C05467=1069.502,171.520,421.573,173.265,27.850,155.032
C05468=1069.508,171.769,421.550,173.266,27.852,155.033
C05469=1069.513,172.019,421.528,173.269,27.855,155.033
C05470=1069.519,172.267,421.505,173.270,27.858,155.034
C05471=1069.525,172.515,421.483,173.273,27.861,155.034
C05472=1069.530,172.765,421.461,173.274,27.864,155.034
C05473=1069.536,173.014,421.438,173.277,27.867,155.035
C05474=1069.542,173.263,421.416,173.278,27.870,155.035
C05475=1069.548,173.512,421.393,173.280,27.872,155.036
C05476=1069.553,173.760,421.370,173.282,27.875,155.036
C05477=1069.558,174.010,421.348,173.284,27.878,155.036
C05478=1069.565,174.258,421.326,173.286,27.881,155.037
C05479=1069.570,174.508,421.304,173.288,27.884,155.037
C05480=1069.576,174.790,421.278,173.290,27.887,155.037
C05481=1069.583,175.072,421.253,173.293,27.890,155.038
C05482=1069.590,175.355,421.226,173.295,27.893,155.038
C05483=1069.597,175.637,421.201,173.297,27.897,155.039
C05484=1069.602,175.886,421.179,173.299,27.900,155.039
C05485=1069.608,176.135,421.156,173.301,27.902,155.040
C05486=1069.614,176.383,421.134,173.303,27.905,155.040
C05487=1069.619,176.633,421.112,173.305,27.908,155.040
C05488=1069.625,176.881,421.089,173.307,27.911,155.041
C05489=1069.631,177.130,421.066,173.309,27.913,155.041
C05490=1069.637,177.379,421.043,173.311,27.916,155.042
C05491=1069.642,177.628,421.021,173.313,27.919,155.042
C05492=1069.648,177.877,420.998,173.315,27.922,155.042
C05493=1069.654,178.126,420.975,173.317,27.925,155.043
C05494=1069.660,178.375,420.952,173.319,27.928,155.043
C05495=1069.666,178.624,420.930,173.321,27.931,155.044
C05496=1069.672,178.873,420.908,173.323,27.933,155.044
C05497=1069.677,179.122,420.885,173.325,27.936,155.044
C05498=1069.682,179.370,420.862,173.327,27.939,155.045
C05499=1069.688,179.619,420.839,173.329,27.942,155.045
C05500=1069.695,179.868,420.817,173.331,27.945,155.046
C05501=1069.700,180.117,420.794,173.333,27.948,155.046
C05502=1069.706,180.366,420.771,173.335,27.950,155.046
C05503=1069.711,180.615,420.749,173.337,27.953,155.047
C05504=1069.717,180.864,420.726,173.339,27.956,155.047
C05505=1069.724,181.113,420.704,173.341,27.959,155.048
C05506=1069.729,181.361,420.681,173.343,27.961,155.048
C05507=1069.735,181.610,420.658,173.345,27.964,155.048
C05508=1069.741,181.859,420.635,173.348,27.967,155.049
C05509=1069.747,182.108,420.612,173.349,27.970,155.049
C05510=1069.753,182.357,420.589,173.352,27.973,155.049
C05511=1069.759,182.606,420.566,173.353,27.976,155.050
C05512=1069.765,182.855,420.544,173.356,27.979,155.050
C05513=1069.770,183.103,420.521,173.357,27.982,155.051
C05514=1069.777,183.353,420.497,173.360,27.985,155.051
C05515=1069.782,183.602,420.474,173.362,27.987,155.051
C05516=1069.788,183.851,420.451,173.364,27.990,155.052
C05517=1069.795,184.099,420.429,173.366,27.993,155.052
C05518=1069.800,184.348,420.406,173.368,27.995,155.052
C05519=1069.806,184.597,420.383,173.370,27.998,155.053
C05520=1069.812,184.846,420.360,173.372,28.001,155.053
C05521=1069.817,185.095,420.337,173.374,28.004,155.054
C05522=1069.822,185.344,420.314,173.376,28.007,155.054
C05523=1069.828,185.593,420.291,173.378,28.010,155.055
C05524=1069.834,185.841,420.267,173.380,28.013,155.055
C05525=1069.839,186.091,420.244,173.382,28.016,155.055
C05526=1069.845,186.339,420.221,173.384,28.019,155.056
C05527=1069.851,186.588,420.198,173.387,28.022,155.056
C05528=1069.856,186.837,420.175,173.388,28.025,155.057
C05529=1069.861,187.087,420.151,173.391,28.028,155.057
C05530=1069.867,187.335,420.128,173.392,28.031,155.057
C05531=1069.873,187.584,420.105,173.395,28.034,155.058
C05532=1069.878,187.833,420.081,173.396,28.037,155.058
C05533=1069.884,188.082,420.058,173.399,28.040,155.059
C05534=1069.890,188.331,420.035,173.400,28.043,155.059
C05535=1069.896,188.579,420.011,173.403,28.046,155.060
C05536=1069.901,188.828,419.988,173.404,28.049,155.060
C05537=1069.906,189.077,419.965,173.407,28.052,155.060
C05538=1069.912,189.325,419.941,173.409,28.055,155.061
C05539=1069.917,189.575,419.918,173.411,28.058,155.061
C05540=1069.923,189.823,419.895,173.413,28.061,155.062
C05541=1069.929,190.072,419.872,173.415,28.063,155.062
C05542=1069.934,190.321,419.848,173.417,28.067,155.063
C05543=1069.940,190.570,419.825,173.419,28.070,155.063
C05544=1069.946,190.852,419.798,173.421,28.073,155.063
C05545=1069.952,191.133,419.772,173.424,28.076,155.064
C05546=1069.959,191.416,419.745,173.426,28.080,155.064
C05547=1069.965,191.698,419.718,173.429,28.083,155.065
C05548=1069.971,191.946,419.695,173.431,28.086,155.065
C05549=1069.977,192.195,419.672,173.433,28.089,155.066
C05550=1069.982,192.444,419.648,173.435,28.092,155.066
C05551=1069.988,192.693,419.624,173.438,28.095,155.066
C05552=1069.994,192.942,419.601,173.439,28.098,155.067
C05553=1069.999,193.191,419.577,173.442,28.101,155.067
C05554=1070.005,193.440,419.554,173.443,28.104,155.068
C05555=1070.011,193.688,419.530,173.446,28.107,155.068
C05556=1070.016,193.937,419.507,173.448,28.110,155.069
C05557=1070.022,194.185,419.483,173.450,28.113,155.069
C05558=1070.027,194.435,419.460,173.452,28.116,155.069
C05559=1070.034,194.684,419.435,173.454,28.119,155.070
C05560=1070.040,194.933,419.413,173.456,28.122,155.070
C05561=1070.045,195.181,419.388,173.459,28.125,155.071
C05562=1070.051,195.430,419.365,173.460,28.128,155.071
C05563=1070.056,195.679,419.341,173.463,28.131,155.072
C05564=1070.062,195.928,419.318,173.464,28.134,155.072
C05565=1070.068,196.176,419.294,173.467,28.137,155.072
C05566=1070.074,196.425,419.270,173.469,28.140,155.073
C05567=1070.079,196.674,419.247,173.471,28.142,155.073
C05568=1070.085,196.923,419.223,173.474,28.145,155.074
C05569=1070.091,197.172,419.199,173.476,28.149,155.074
C05570=1070.097,197.420,419.176,173.478,28.152,155.074
C05571=1070.102,197.669,419.151,173.480,28.155,155.075
C05572=1070.108,197.918,419.128,173.483,28.158,155.075
C05573=1070.114,198.167,419.104,173.484,28.160,155.076
C05574=1070.120,198.415,419.080,173.487,28.163,155.076
C05575=1070.125,198.665,419.057,173.488,28.167,155.077
C05576=1070.131,198.913,419.033,173.491,28.170,155.077
C05577=1070.137,199.162,419.008,173.493,28.173,155.077
C05578=1070.143,199.411,418.985,173.495,28.175,155.078
C05579=1070.149,199.659,418.962,173.497,28.178,155.078
C05580=1070.154,199.909,418.937,173.500,28.181,155.079
C05581=1070.161,200.157,418.913,173.501,28.184,155.079
C05582=1070.166,200.406,418.889,173.504,28.187,155.079
C05583=1070.172,200.655,418.866,173.506,28.190,155.080
C05584=1070.177,200.904,418.842,173.508,28.193,155.080
C05585=1070.183,201.152,418.818,173.510,28.196,155.081
C05586=1070.189,201.401,418.793,173.513,28.200,155.081
C05587=1070.195,201.650,418.770,173.515,28.203,155.082
C05588=1070.200,201.899,418.746,173.517,28.205,155.082
C05589=1070.207,202.148,418.722,173.519,28.208,155.082
C05590=1070.212,202.396,418.698,173.522,28.211,155.083
C05591=1070.218,202.645,418.674,173.523,28.214,155.083
C05592=1070.224,202.894,418.650,173.526,28.217,155.084
C05593=1070.230,203.143,418.625,173.528,28.220,155.084
C05594=1070.235,203.391,418.601,173.530,28.224,155.085
C05595=1070.241,203.639,418.577,173.533,28.227,155.085
C05596=1070.247,203.889,418.554,173.535,28.230,155.085
C05597=1070.252,204.138,418.529,173.537,28.233,155.086
C05598=1070.257,204.386,418.505,173.539,28.236,155.086
C05599=1070.264,204.635,418.481,173.542,28.239,155.087
C05600=1070.269,204.884,418.457,173.543,28.242,155.087
C05601=1070.274,205.133,418.432,173.546,28.245,155.088
C05602=1070.280,205.382,418.408,173.548,28.248,155.088
C05603=1070.286,205.630,418.384,173.551,28.251,155.088
C05604=1070.292,205.879,418.360,173.552,28.254,155.089
C05605=1070.297,206.128,418.335,173.555,28.258,155.089
C05606=1070.303,206.377,418.311,173.557,28.261,155.090
C05607=1070.309,206.625,418.286,173.559,28.263,155.090
C05608=1070.338,207.881,418.163,173.698,28.338,155.093
C05609=1070.343,208.093,418.142,173.701,28.341,155.094
C05610=1070.348,208.306,418.120,173.702,28.344,155.094
C05611=1070.353,208.518,418.099,173.704,28.348,155.095
C05612=1070.359,208.731,418.077,173.705,28.352,155.096
C05613=1070.363,208.944,418.056,173.707,28.355,155.096
C05614=1070.368,209.156,418.034,173.709,28.358,155.097
C05615=1070.373,209.369,418.013,173.710,28.361,155.097
C05616=1070.379,209.618,417.988,173.713,28.366,155.098
C05617=1070.385,209.866,417.963,173.714,28.369,155.099
C05618=1070.391,210.115,417.938,173.717,28.373,155.099
C05619=1070.397,210.364,417.913,173.719,28.378,155.100
C05620=1070.402,210.612,417.887,173.720,28.382,155.101
C05621=1070.409,210.861,417.862,173.723,28.386,155.101
C05622=1070.414,211.110,417.837,173.725,28.390,155.102
C05623=1070.420,211.358,417.812,173.726,28.394,155.103
C05624=1070.426,211.607,417.787,173.729,28.398,155.103
C05625=1070.432,211.856,417.761,173.731,28.402,155.104
C05626=1070.437,212.104,417.736,173.733,28.405,155.104
C05627=1070.444,212.353,417.711,173.735,28.410,155.105
C05628=1070.449,212.602,417.686,173.737,28.414,155.106
C05629=1070.456,212.851,417.661,173.739,28.417,155.106
C05630=1070.461,213.099,417.635,173.741,28.421,155.107
C05631=1070.467,213.348,417.610,173.744,28.425,155.108
C05632=1070.473,213.596,417.584,173.745,28.430,155.108
C05633=1070.478,213.845,417.558,173.747,28.434,155.109
C05634=1070.484,214.093,417.533,173.750,28.438,155.110
C05635=1070.490,214.342,417.508,173.751,28.442,155.110
C05636=1070.496,214.591,417.482,173.754,28.446,155.111
C05637=1070.502,214.840,417.457,173.756,28.450,155.112
C05638=1070.508,215.088,417.432,173.757,28.453,155.112
C05639=1070.513,215.336,417.406,173.760,28.457,155.113
C05640=1070.519,215.585,417.381,173.762,28.462,155.114
C05641=1070.525,215.834,417.355,173.764,28.465,155.114
C05642=1070.531,216.083,417.329,173.766,28.469,155.115
C05643=1070.537,216.331,417.304,173.768,28.474,155.116
C05644=1070.543,216.580,417.278,173.770,28.478,155.116
C05645=1070.548,216.828,417.253,173.772,28.482,155.117
C05646=1070.554,217.077,417.228,173.775,28.486,155.118
C05647=1070.560,217.326,417.202,173.776,28.490,155.118
C05648=1070.566,217.575,417.176,173.778,28.494,155.119
C05649=1070.572,217.823,417.150,173.781,28.498,155.119
C05650=1070.578,218.072,417.125,173.783,28.502,155.120
C05651=1070.584,218.320,417.099,173.785,28.505,155.121
C05652=1070.590,218.569,417.073,173.787,28.509,155.121
C05653=1070.595,218.817,417.048,173.789,28.513,155.122
C05654=1070.601,219.066,417.022,173.791,28.517,155.123
C05655=1070.607,219.314,416.996,173.793,28.521,155.123
C05656=1070.613,219.563,416.971,173.796,28.525,155.124
C05657=1070.619,219.812,416.945,173.798,28.529,155.125
C05658=1070.625,220.061,416.920,173.799,28.533,155.125
C05659=1070.631,220.310,416.894,173.802,28.537,155.126
C05660=1070.637,220.558,416.868,173.804,28.541,155.127
C05661=1070.643,220.807,416.842,173.806,28.545,155.127
C05662=1070.649,221.055,416.816,173.808,28.549,155.128
C05663=1070.655,221.304,416.791,173.811,28.553,155.129
C05664=1070.660,221.519,416.768,173.812,28.556,155.129
C05665=1070.665,221.733,416.746,173.815,28.560,155.130
C05666=1070.670,221.948,416.723,173.816,28.563,155.130
C05667=1070.675,222.163,416.702,173.817,28.567,155.131
C05668=1070.680,222.379,416.678,173.820,28.570,155.131
C05669=1070.685,222.593,416.656,173.821,28.573,155.132
C05670=1070.690,222.808,416.633,173.823,28.577,155.132
C05671=1070.695,223.022,416.611,173.825,28.580,155.133
C05672=1070.701,223.271,416.585,173.827,28.584,155.134
C05673=1070.707,223.520,416.560,173.829,28.588,155.134
C05674=1070.713,223.768,416.533,173.832,28.592,155.135
C05675=1070.718,224.017,416.507,173.834,28.596,155.136
C05676=1070.725,224.265,416.481,173.836,28.600,155.136
C05677=1070.730,224.514,416.455,173.838,28.604,155.137
C05678=1070.736,224.763,416.429,173.840,28.608,155.138
C05679=1070.741,225.012,416.403,173.843,28.612,155.138
C05680=1070.748,225.260,416.377,173.844,28.616,155.139
C05681=1070.753,225.509,416.351,173.847,28.620,155.139
C05682=1070.759,225.757,416.324,173.849,28.624,155.140
C05683=1070.765,226.006,416.299,173.851,28.628,155.141
C05684=1070.771,226.254,416.272,173.853,28.632,155.141
C05685=1070.776,226.503,416.246,173.855,28.636,155.142
C05686=1070.783,226.751,416.220,173.858,28.640,155.143
C05687=1070.788,227.000,416.194,173.860,28.644,155.143
C05688=1070.794,227.248,416.167,173.862,28.648,155.144
C05689=1070.800,227.497,416.141,173.864,28.652,155.145
C05690=1070.806,227.745,416.115,173.866,28.656,155.145
C05691=1070.812,227.994,416.089,173.869,28.659,155.146
C05692=1070.817,228.243,416.063,173.870,28.663,155.146
C05693=1070.825,228.492,416.036,173.873,28.667,155.147
C05694=1070.830,228.740,416.010,173.875,28.671,155.148
C05695=1070.836,228.989,415.984,173.878,28.675,155.148
C05696=1070.842,229.237,415.957,173.880,28.679,155.149
C05697=1070.848,229.485,415.931,173.882,28.683,155.150
C05698=1070.854,229.734,415.905,173.884,28.687,155.150
C05699=1070.859,229.983,415.879,173.886,28.691,155.151
C05700=1070.865,230.231,415.852,173.889,28.695,155.152
C05701=1070.871,230.480,415.825,173.891,28.699,155.152
C05702=1070.877,230.729,415.799,173.893,28.702,155.153
C05703=1070.883,230.977,415.772,173.895,28.706,155.154
C05704=1070.888,231.226,415.746,173.898,28.710,155.154
C05705=1070.894,231.474,415.719,173.900,28.714,155.155
C05706=1070.901,231.722,415.693,173.901,28.718,155.155
C05707=1070.906,231.971,415.667,173.904,28.722,155.156
C05708=1070.912,232.220,415.640,173.906,28.726,155.157
C05709=1070.918,232.469,415.613,173.909,28.730,155.157
C05710=1070.924,232.717,415.587,173.911,28.734,155.158
C05711=1070.930,232.965,415.560,173.913,28.738,155.159
C05712=1070.936,233.214,415.533,173.915,28.742,155.159
C05713=1070.941,233.462,415.507,173.917,28.746,155.160
C05714=1070.947,233.710,415.480,173.920,28.750,155.161
C05715=1070.953,233.960,415.454,173.922,28.754,155.161
C05716=1070.959,234.208,415.427,173.925,28.758,155.162
C05717=1070.965,234.457,415.401,173.926,28.762,155.163
C05718=1070.971,234.705,415.374,173.929,28.766,155.163
C05719=1070.976,234.954,415.347,173.931,28.770,155.164
C05720=1070.981,235.165,415.324,173.933,28.773,155.164
C05721=1070.986,235.375,415.302,173.935,28.776,155.165
C05722=1070.991,235.586,415.278,173.937,28.779,155.165
C05723=1070.996,235.797,415.256,173.939,28.783,155.166
C05724=1071.001,236.008,415.233,173.941,28.787,155.167
C05725=1071.006,236.219,415.211,173.942,28.790,155.167
C05726=1071.011,236.429,415.188,173.945,28.793,155.168
C05727=1071.016,236.640,415.164,173.946,28.796,155.168
C05728=1071.022,236.888,415.138,173.949,28.800,155.169
C05729=1071.028,237.136,415.111,173.951,28.804,155.170
C05730=1071.033,237.385,415.084,173.954,28.808,155.170
C05731=1071.040,237.634,415.057,173.955,28.812,155.171
C05732=1071.045,237.882,415.031,173.957,28.816,155.172
C05733=1071.050,238.131,415.003,173.960,28.820,155.172
C05734=1071.057,238.380,414.976,173.962,28.824,155.173
C05735=1071.063,238.628,414.949,173.965,28.828,155.173
C05736=1071.069,238.876,414.922,173.967,28.832,155.174
C05737=1071.074,239.124,414.896,173.970,28.835,155.175
C05738=1071.081,239.374,414.869,173.971,28.839,155.175
C05739=1071.087,239.622,414.842,173.974,28.843,155.176
C05740=1071.092,239.870,414.814,173.976,28.847,155.177
C05741=1071.098,240.119,414.787,173.979,28.851,155.177
C05742=1071.104,240.367,414.760,173.981,28.855,155.178
C05743=1071.110,240.616,414.734,173.983,28.859,155.178
C05744=1071.117,240.864,414.706,173.986,28.863,155.179
C05745=1071.122,241.113,414.679,173.987,28.867,155.180
C05746=1071.127,241.361,414.652,173.990,28.871,155.180
C05747=1071.134,241.610,414.624,173.992,28.875,155.181
C05748=1071.140,241.858,414.598,173.995,28.879,155.182
C05749=1071.146,242.106,414.571,173.997,28.883,155.182
C05750=1071.152,242.355,414.543,174.000,28.887,155.183
C05751=1071.157,242.603,414.516,174.002,28.890,155.184
C05752=1071.163,242.851,414.489,174.005,28.894,155.184
C05753=1071.169,243.101,414.461,174.006,28.898,155.185
C05754=1071.175,243.349,414.435,174.009,28.902,155.185
C05755=1071.180,243.597,414.407,174.011,28.906,155.186
C05756=1071.187,243.846,414.380,174.013,28.910,155.187
C05757=1071.193,244.094,414.352,174.016,28.914,155.188
C05758=1071.198,244.342,414.325,174.018,28.918,155.188
C05759=1071.204,244.591,414.297,174.021,28.922,155.189
C05760=1071.209,244.840,414.270,174.023,28.926,155.189
C05761=1071.216,245.088,414.242,174.026,28.930,155.190
C05762=1071.221,245.337,414.215,174.027,28.934,155.191
C05763=1071.227,245.584,414.188,174.030,28.938,155.191
C05764=1071.234,245.833,414.161,174.032,28.941,155.192
C05765=1071.239,246.082,414.133,174.035,28.945,155.193
C05766=1071.246,246.330,414.105,174.037,28.949,155.193
C05767=1071.251,246.579,414.078,174.039,28.953,155.194
C05768=1071.257,246.827,414.050,174.042,28.957,155.194
C05769=1071.262,247.076,414.023,174.044,28.961,155.195
C05770=1071.268,247.324,413.995,174.047,28.966,155.196
C05771=1071.274,247.572,413.967,174.049,28.970,155.197
C05772=1071.279,247.821,413.940,174.051,28.973,155.197
C05773=1071.285,248.069,413.912,174.053,28.977,155.198
C05774=1071.291,248.317,413.884,174.056,28.981,155.199
C05775=1071.297,248.565,413.856,174.058,28.985,155.199
C05776=1071.306,248.981,413.811,174.062,28.992,155.200
C05777=1071.316,249.396,413.763,174.066,28.999,155.201
C05778=1071.326,249.811,413.717,174.070,29.005,155.202
C05779=1071.335,250.226,413.671,174.074,29.012,155.204
C05780=1071.341,250.474,413.643,174.077,29.016,155.204
C05781=1071.347,250.723,413.615,174.079,29.020,155.205
C05782=1071.353,250.971,413.588,174.082,29.024,155.206
C05783=1071.359,251.220,413.559,174.084,29.028,155.206
C05784=1071.365,251.467,413.532,174.086,29.032,155.207
C05785=1071.371,251.716,413.504,174.088,29.036,155.207
C05786=1071.376,251.965,413.476,174.091,29.040,155.208
C05787=1071.382,252.213,413.449,174.093,29.044,155.209
C05788=1071.388,252.461,413.421,174.096,29.048,155.209
C05789=1071.394,252.710,413.392,174.098,29.052,155.210
C05790=1071.399,252.958,413.364,174.101,29.056,155.211
C05791=1071.406,253.207,413.337,174.103,29.060,155.211
C05792=1071.412,253.455,413.308,174.106,29.064,155.212
C05793=1071.417,253.703,413.280,174.108,29.067,155.213
C05794=1071.423,253.952,413.252,174.111,29.071,155.213
C05795=1071.429,254.200,413.225,174.113,29.075,155.214
C05796=1071.435,254.449,413.196,174.115,29.079,155.215
C05797=1071.440,254.697,413.168,174.118,29.083,155.215
C05798=1071.446,254.945,413.140,174.120,29.087,155.216
C05799=1071.453,255.194,413.112,174.123,29.091,155.217
C05800=1071.458,255.442,413.084,174.125,29.095,155.217
C05801=1071.464,255.691,413.056,174.128,29.099,155.218
C05802=1071.470,255.938,413.027,174.130,29.103,155.218
C05803=1071.476,256.186,413.000,174.133,29.107,155.219
C05804=1071.482,256.435,412.971,174.135,29.111,155.220
C05805=1071.488,256.683,412.943,174.138,29.115,155.220
C05806=1071.494,256.932,412.915,174.140,29.119,155.221
C05807=1071.500,257.181,412.887,174.143,29.123,155.222
C05808=1071.506,257.429,412.859,174.145,29.127,155.222
C05809=1071.512,257.677,412.830,174.148,29.131,155.223
C05810=1071.518,257.925,412.802,174.150,29.135,155.224
C05811=1071.523,258.173,412.774,174.153,29.138,155.224
C05812=1071.529,258.422,412.746,174.155,29.142,155.225
C05813=1071.535,258.670,412.717,174.158,29.146,155.225
C05814=1071.541,258.918,412.689,174.160,29.150,155.226
C05815=1071.547,259.167,412.661,174.163,29.154,155.227
C05816=1071.553,259.416,412.633,174.165,29.158,155.227
C05817=1071.560,259.664,412.604,174.168,29.162,155.228
C05818=1071.565,259.912,412.576,174.170,29.166,155.229
C05819=1071.571,260.161,412.547,174.173,29.170,155.229
C05820=1071.578,260.408,412.519,174.175,29.173,155.230
C05821=1071.584,260.657,412.490,174.178,29.177,155.231
C05822=1071.589,260.905,412.463,174.180,29.181,155.231
C05823=1071.595,261.153,412.433,174.183,29.185,155.232
C05824=1071.601,261.402,412.405,174.185,29.189,155.233
C05825=1071.608,261.650,412.376,174.187,29.193,155.233
C05826=1071.614,261.899,412.348,174.190,29.197,155.234
C05827=1071.620,262.147,412.320,174.193,29.200,155.234
C05828=1071.630,262.559,412.273,174.197,29.207,155.235
C05829=1071.640,262.971,412.225,174.201,29.214,155.237
C05830=1071.651,263.385,412.178,174.205,29.220,155.238
C05831=1071.661,263.797,412.130,174.209,29.227,155.239
C05832=1071.665,264.045,412.101,174.212,29.231,155.239
C05833=1071.671,264.294,412.073,174.214,29.235,155.240
C05834=1071.678,264.542,412.044,174.217,29.239,155.241
C05835=1071.684,264.791,412.015,174.219,29.242,155.241
C05836=1071.690,265.039,411.986,174.223,29.247,155.242
C05837=1071.695,265.286,411.957,174.225,29.251,155.243
C05838=1071.701,265.535,411.929,174.228,29.254,155.243
C05839=1071.707,265.783,411.900,174.230,29.258,155.244
C05840=1071.713,266.031,411.871,174.233,29.262,155.245
C05841=1071.719,266.280,411.842,174.235,29.266,155.245
C05842=1071.725,266.528,411.814,174.238,29.270,155.246
C05843=1071.730,266.776,411.784,174.240,29.274,155.246
C05844=1071.736,267.025,411.756,174.243,29.278,155.247
C05845=1071.743,267.273,411.727,174.245,29.282,155.248
C05846=1071.749,267.521,411.698,174.248,29.286,155.249
C05847=1071.754,267.769,411.668,174.250,29.290,155.249
C05848=1071.760,268.018,411.640,174.253,29.294,155.250
C05849=1071.766,268.266,411.611,174.255,29.298,155.251
C05850=1071.772,268.514,411.582,174.258,29.302,155.251
C05851=1071.778,268.762,411.553,174.261,29.306,155.252
C05852=1071.784,269.010,411.523,174.264,29.310,155.252
C05853=1071.790,269.258,411.494,174.266,29.314,155.253
C05854=1071.796,269.507,411.466,174.269,29.318,155.254
C05855=1071.802,269.756,411.436,174.271,29.322,155.254
C05856=1071.808,270.004,411.407,174.274,29.326,155.255
C05857=1071.814,270.252,411.378,174.276,29.330,155.256
C05858=1071.819,270.500,411.349,174.279,29.334,155.256
C05859=1071.825,270.748,411.320,174.281,29.338,155.257
C05860=1071.831,270.996,411.291,174.284,29.342,155.258
C05861=1071.837,271.244,411.261,174.286,29.346,155.258
C05862=1071.843,271.493,411.232,174.290,29.350,155.259
C05863=1071.849,271.741,411.202,174.292,29.354,155.260
C05864=1071.855,271.989,411.173,174.295,29.358,155.260
C05865=1071.861,272.237,411.144,174.297,29.362,155.261
C05866=1071.867,272.486,411.115,174.300,29.366,155.262
C05867=1071.873,272.734,411.086,174.302,29.370,155.262
C05868=1071.879,272.982,411.056,174.305,29.374,155.263
C05869=1071.885,273.230,411.027,174.307,29.378,155.264
C05870=1071.891,273.479,410.998,174.310,29.382,155.264
C05871=1071.897,273.727,410.968,174.313,29.386,155.265
C05872=1071.903,273.974,410.939,174.316,29.390,155.266
C05873=1071.909,274.223,410.909,174.318,29.394,155.266
C05874=1071.915,274.471,410.880,174.321,29.398,155.267
C05875=1071.920,274.719,410.850,174.323,29.402,155.268
C05876=1071.926,274.968,410.821,174.326,29.406,155.268
C05877=1071.932,275.216,410.792,174.328,29.410,155.269
C05878=1071.938,275.464,410.761,174.332,29.414,155.270
C05879=1071.944,275.712,410.732,174.334,29.418,155.270
C05880=1071.953,276.128,410.683,174.338,29.425,155.271
C05881=1071.964,276.544,410.633,174.342,29.432,155.273
C05882=1071.973,276.959,410.583,174.347,29.438,155.274
C05883=1071.983,277.375,410.534,174.352,29.445,155.275
C05884=1071.989,277.623,410.504,174.354,29.449,155.276
C05885=1071.995,277.871,410.475,174.357,29.453,155.276
C05886=1072.001,278.120,410.445,174.359,29.457,155.277
C05887=1072.007,278.368,410.414,174.362,29.461,155.278
C05888=1072.014,278.616,410.385,174.365,29.465,155.278
C05889=1072.019,278.864,410.355,174.368,29.470,155.279
C05890=1072.025,279.113,410.325,174.370,29.474,155.280
C05891=1072.031,279.361,410.296,174.373,29.477,155.280
C05892=1072.037,279.609,410.266,174.375,29.481,155.281
C05893=1072.043,279.857,410.236,174.378,29.485,155.282
C05894=1072.049,280.105,410.207,174.381,29.490,155.282
C05895=1072.055,280.353,410.177,174.384,29.494,155.283
C05896=1072.061,280.602,410.146,174.386,29.498,155.284
C05897=1072.067,280.850,410.117,174.389,29.502,155.284
C05898=1072.073,281.098,410.087,174.391,29.506,155.285
C05899=1072.079,281.345,410.057,174.394,29.510,155.286
C05900=1072.084,281.594,410.027,174.397,29.514,155.286
C05901=1072.090,281.842,409.997,174.400,29.518,155.287
C05902=1072.096,282.090,409.967,174.402,29.522,155.288
C05903=1072.102,282.338,409.937,174.405,29.526,155.288
C05904=1072.109,282.586,409.906,174.408,29.530,155.289
C05905=1072.114,282.835,409.877,174.411,29.535,155.290
C05906=1072.120,283.082,409.846,174.414,29.539,155.290
C05907=1072.126,283.330,409.816,174.416,29.543,155.291
C05908=1072.131,283.579,409.786,174.419,29.546,155.292
C05909=1072.137,283.826,409.756,174.421,29.551,155.293
C05910=1072.144,284.075,409.725,174.425,29.555,155.293
C05911=1072.149,284.323,409.695,174.427,29.559,155.294
C05912=1072.155,284.571,409.665,174.430,29.563,155.295
C05913=1072.162,284.819,409.636,174.432,29.567,155.295
C05914=1072.167,285.067,409.605,174.436,29.571,155.296
C05915=1072.174,285.315,409.575,174.438,29.576,155.297
C05916=1072.180,285.563,409.544,174.441,29.580,155.297
C05917=1072.185,285.811,409.515,174.443,29.583,155.298
C05918=1072.191,286.059,409.484,174.446,29.587,155.299
C05919=1072.197,286.308,409.454,174.449,29.592,155.299
C05920=1072.203,286.555,409.423,174.452,29.596,155.300
C05921=1072.209,286.803,409.393,174.454,29.600,155.301
C05922=1072.215,287.051,409.362,174.457,29.604,155.302
C05923=1072.221,287.300,409.332,174.460,29.608,155.302
C05924=1072.227,287.547,409.301,174.463,29.612,155.303
C05925=1072.233,287.795,409.271,174.465,29.617,155.304
C05926=1072.239,288.044,409.240,174.468,29.620,155.304
C05927=1072.246,288.291,409.211,174.471,29.625,155.305
C05928=1072.252,288.539,409.180,174.474,29.628,155.306
C05929=1072.257,288.787,409.150,174.476,29.633,155.306
C05930=1072.264,289.035,409.119,174.479,29.637,155.307
C05931=1072.269,289.284,409.088,174.483,29.641,155.308
C05932=1072.274,289.497,409.063,174.484,29.644,155.308
C05933=1072.279,289.710,409.036,174.487,29.648,155.309
C05934=1072.285,289.923,409.010,174.489,29.652,155.310
C05935=1072.289,290.136,408.984,174.492,29.655,155.310
C05936=1072.295,290.349,408.957,174.494,29.659,155.311
C05937=1072.300,290.562,408.931,174.496,29.662,155.311
C05938=1072.305,290.774,408.905,174.499,29.666,155.312
C05939=1072.310,290.989,408.878,174.501,29.669,155.312
C05940=1072.316,291.236,408.847,174.504,29.674,155.313
C05941=1072.322,291.484,408.817,174.507,29.678,155.314
C05942=1072.328,291.732,408.786,174.510,29.682,155.315
C05943=1072.334,291.980,408.756,174.512,29.686,155.315
C05944=1072.340,292.228,408.725,174.515,29.690,155.316
C05945=1072.346,292.476,408.693,174.518,29.694,155.317
C05946=1072.352,292.724,408.663,174.521,29.698,155.317
C05947=1072.358,292.972,408.632,174.523,29.703,155.318
C05948=1072.364,293.219,408.601,174.527,29.707,155.319
C05949=1072.369,293.468,408.570,174.529,29.711,155.320
C05950=1072.376,293.716,408.540,174.532,29.715,155.320
C05951=1072.381,293.964,408.509,174.535,29.720,155.321
C05952=1072.388,294.212,408.478,174.538,29.724,155.322
C05953=1072.394,294.460,408.447,174.541,29.728,155.322
C05954=1072.400,294.708,408.415,174.543,29.732,155.323
C05955=1072.406,294.956,408.385,174.547,29.736,155.324
C05956=1072.412,295.204,408.355,174.549,29.740,155.325
C05957=1072.418,295.452,408.323,174.552,29.745,155.325
C05958=1072.423,295.700,408.292,174.555,29.749,155.326
C05959=1072.430,295.947,408.261,174.558,29.753,155.327
C05960=1072.435,296.196,408.230,174.560,29.757,155.327
C05961=1072.442,296.444,408.199,174.564,29.762,155.328
C05962=1072.448,296.691,408.168,174.566,29.766,155.329
C05963=1072.454,296.940,408.136,174.569,29.770,155.330
C05964=1072.460,297.187,408.106,174.572,29.774,155.330
C05965=1072.466,297.435,408.074,174.575,29.778,155.331
C05966=1072.471,297.683,408.043,174.577,29.782,155.332
C05967=1072.477,297.932,408.011,174.581,29.787,155.332
C05968=1072.484,298.179,407.980,174.583,29.791,155.333
C05969=1072.489,298.427,407.949,174.586,29.796,155.334
C05970=1072.495,298.675,407.918,174.590,29.800,155.335
C05971=1072.501,298.922,407.886,174.592,29.804,155.335
C05972=1072.506,299.171,407.855,174.595,29.808,155.336
C05973=1072.513,299.418,407.824,174.598,29.813,155.337
C05974=1072.519,299.667,407.792,174.601,29.817,155.338
C05975=1072.524,299.915,407.761,174.603,29.821,155.338
C05976=1072.530,300.163,407.729,174.607,29.826,155.339
C05977=1072.536,300.410,407.698,174.609,29.830,155.340
C05978=1072.542,300.658,407.666,174.612,29.834,155.341
C05979=1072.548,300.906,407.635,174.615,29.839,155.341
C05980=1072.553,301.154,407.603,174.618,29.843,155.342
C05981=1072.560,301.402,407.572,174.621,29.847,155.343
C05982=1072.566,301.650,407.540,174.624,29.852,155.344
C05983=1072.571,301.897,407.509,174.626,29.856,155.344
C05984=1072.578,302.145,407.477,174.630,29.861,155.345
C05985=1072.583,302.393,407.446,174.632,29.864,155.346
C05986=1072.589,302.641,407.414,174.635,29.869,155.347
C05987=1072.595,302.890,407.382,174.638,29.873,155.347
C05988=1072.600,303.109,407.354,174.641,29.877,155.348
C05989=1072.606,303.330,407.327,174.644,29.881,155.349
C05990=1072.611,303.550,407.298,174.646,29.885,155.349
C05991=1072.616,303.771,407.270,174.649,29.889,155.350
C05992=1072.621,303.991,407.241,174.651,29.893,155.351
C05993=1072.627,304.211,407.213,174.654,29.896,155.351
C05994=1072.632,304.431,407.185,174.657,29.900,155.352
C05995=1072.637,304.651,407.157,174.659,29.904,155.353
C05996=1072.643,304.900,407.125,174.662,29.908,155.353
C05997=1072.650,305.148,407.093,174.665,29.913,155.354
C05998=1072.655,305.395,407.062,174.668,29.917,155.355
C05999=1072.661,305.643,407.030,174.671,29.921,155.356
C06000=1072.667,305.892,406.998,174.674,29.926,155.356
C06001=1072.673,306.139,406.966,174.677,29.930,155.357
C06002=1072.679,306.387,406.934,174.680,29.935,155.358
C06003=1072.685,306.635,406.902,174.682,29.939,155.359
C06004=1072.691,306.882,406.870,174.686,29.943,155.359
C06005=1072.698,307.130,406.839,174.689,29.948,155.360
C06006=1072.704,307.378,406.807,174.692,29.952,155.361
C06007=1072.710,307.626,406.775,174.695,29.957,155.362
C06008=1072.715,307.874,406.743,174.698,29.961,155.362
C06009=1072.722,308.121,406.711,174.701,29.965,155.363
C06010=1072.728,308.369,406.679,174.704,29.969,155.364
C06011=1072.734,308.618,406.647,174.707,29.974,155.365
C06012=1072.740,308.866,406.615,174.709,29.978,155.366
C06013=1072.746,309.113,406.582,174.713,29.983,155.366
C06014=1072.753,309.361,406.551,174.715,29.987,155.367
C06015=1072.759,309.609,406.519,174.719,29.991,155.368
C06016=1072.765,309.856,406.486,174.721,29.996,155.369
C06017=1072.771,310.105,406.454,174.725,30.000,155.369
C06018=1072.776,310.352,406.422,174.728,30.004,155.370
C06019=1072.783,310.599,406.390,174.731,30.009,155.371
C06020=1072.789,310.848,406.358,174.734,30.013,155.371
C06021=1072.796,311.095,406.325,174.737,30.017,155.372
C06022=1072.802,311.343,406.293,174.740,30.022,155.373
C06023=1072.808,311.592,406.261,174.743,30.026,155.374
C06024=1072.814,311.839,406.229,174.746,30.031,155.375
C06025=1072.820,312.087,406.197,174.749,30.035,155.375
C06026=1072.827,312.335,406.164,174.752,30.040,155.376
C06027=1072.832,312.582,406.133,174.755,30.044,155.377
C06028=1072.838,312.830,406.100,174.758,30.048,155.378
C06029=1072.844,313.078,406.068,174.762,30.053,155.378
C06030=1072.851,313.326,406.035,174.764,30.057,155.379
C06031=1072.857,313.573,406.003,174.768,30.061,155.380
C06032=1072.863,313.821,405.971,174.770,30.066,155.381
C06033=1072.869,314.069,405.938,174.774,30.070,155.381
C06034=1072.875,314.317,405.906,174.776,30.075,155.382
C06035=1072.882,314.565,405.873,174.780,30.079,155.383
C06036=1072.888,314.812,405.840,174.782,30.084,155.384
C06037=1072.894,315.061,405.808,174.786,30.088,155.385
C06038=1072.899,315.309,405.775,174.788,30.093,155.386
C06039=1072.906,315.556,405.742,174.792,30.098,155.386
C06040=1072.912,315.804,405.709,174.795,30.102,155.387
C06041=1072.917,316.052,405.677,174.798,30.106,155.388
C06042=1072.923,316.299,405.644,174.801,30.111,155.389
C06043=1072.929,316.547,405.612,174.804,30.116,155.390
C06044=1072.934,316.769,405.582,174.807,30.120,155.390
C06045=1072.940,316.991,405.552,174.809,30.124,155.391
C06046=1072.945,317.213,405.524,174.812,30.128,155.392
C06047=1072.950,317.435,405.494,174.815,30.132,155.392
C06048=1072.955,317.657,405.464,174.817,30.137,155.393
C06049=1072.961,317.879,405.435,174.820,30.140,155.394
C06050=1072.966,318.101,405.406,174.823,30.145,155.395
C06051=1072.972,318.324,405.376,174.826,30.149,155.395
C06052=1072.978,318.571,405.343,174.828,30.154,155.396
C06053=1072.984,318.819,405.309,174.832,30.158,155.397
C06054=1072.990,319.067,405.277,174.835,30.162,155.398
C06055=1072.996,319.314,405.244,174.838,30.168,155.399
C06056=1073.002,319.562,405.211,174.841,30.172,155.400
C06057=1073.008,319.810,405.178,174.844,30.176,155.400
C06058=1073.014,320.058,405.145,174.848,30.181,155.401
C06059=1073.020,320.305,405.112,174.850,30.186,155.402
C06060=1073.026,320.553,405.079,174.854,30.190,155.403
C06061=1073.032,320.801,405.046,174.856,30.195,155.404
C06062=1073.038,321.049,405.013,174.860,30.200,155.404
C06063=1073.044,321.296,404.980,174.862,30.204,155.405
C06064=1073.050,321.544,404.947,174.866,30.209,155.406
C06065=1073.056,321.792,404.914,174.869,30.213,155.407
C06066=1073.062,322.040,404.881,174.872,30.219,155.408
C06067=1073.069,322.287,404.847,174.876,30.223,155.409
C06068=1073.075,322.535,404.814,174.878,30.227,155.409
C06069=1073.081,322.783,404.781,174.882,30.232,155.410
C06070=1073.087,323.031,404.748,174.884,30.237,155.411
C06071=1073.093,323.278,404.715,174.888,30.242,155.412
C06072=1073.099,323.526,404.681,174.891,30.246,155.413
C06073=1073.105,323.773,404.648,174.894,30.251,155.414
C06074=1073.111,324.022,404.614,174.897,30.256,155.414
C06075=1073.117,324.269,404.582,174.900,30.261,155.415
C06076=1073.123,324.517,404.548,174.904,30.265,155.416
C06077=1073.130,324.764,404.515,174.907,30.270,155.417
C06078=1073.135,325.012,404.481,174.910,30.274,155.418
C06079=1073.142,325.260,404.448,174.913,30.279,155.419
C06080=1073.148,325.508,404.414,174.916,30.284,155.419
C06081=1073.155,325.755,404.381,174.919,30.288,155.420
C06082=1073.160,326.003,404.348,174.923,30.293,155.421
C06083=1073.167,326.251,404.314,174.925,30.298,155.422
C06084=1073.173,326.498,404.280,174.929,30.303,155.423
C06085=1073.178,326.746,404.247,174.933,30.307,155.424
C06086=1073.186,326.994,404.213,174.935,30.312,155.425
C06087=1073.191,327.242,404.180,174.939,30.317,155.425
C06088=1073.198,327.489,404.146,174.942,30.322,155.426
C06089=1073.204,327.737,404.113,174.945,30.326,155.427
C06090=1073.210,327.984,404.079,174.948,30.331,155.428
C06091=1073.216,328.232,404.046,174.951,30.336,155.429
C06092=1073.223,328.480,404.012,174.955,30.340,155.430
C06093=1073.229,328.727,403.978,174.958,30.345,155.431
C06094=1073.235,328.975,403.945,174.961,30.350,155.431
C06095=1073.242,329.223,403.911,174.964,30.355,155.432
C06096=1073.247,329.471,403.878,174.968,30.360,155.433
C06097=1073.255,329.718,403.844,174.970,30.364,155.434
C06098=1073.260,329.965,403.810,174.974,30.369,155.435
C06099=1073.266,330.213,403.776,174.977,30.374,155.436
C06100=1073.272,330.432,403.747,174.980,30.378,155.436
C06101=1073.278,330.651,403.716,174.983,30.382,155.437
C06102=1073.284,330.870,403.686,174.986,30.387,155.438
C06103=1073.289,331.089,403.657,174.989,30.391,155.439
C06104=1073.295,331.308,403.627,174.992,30.395,155.439
C06105=1073.300,331.527,403.597,174.994,30.399,155.440
C06106=1073.306,331.745,403.567,174.998,30.404,155.441
C06107=1073.311,331.964,403.536,175.000,30.408,155.442
C06108=1073.317,332.212,403.503,175.004,30.413,155.443
C06109=1073.323,332.460,403.469,175.006,30.418,155.444
C06110=1073.329,332.707,403.435,175.010,30.423,155.445
C06111=1073.336,332.955,403.400,175.014,30.428,155.445
C06112=1073.341,333.202,403.366,175.016,30.433,155.446
C06113=1073.347,333.450,403.332,175.020,30.438,155.447
C06114=1073.354,333.698,403.298,175.023,30.443,155.448
C06115=1073.360,333.945,403.264,175.027,30.448,155.449
C06116=1073.366,334.193,403.229,175.029,30.452,155.450
C06117=1073.372,334.440,403.195,175.033,30.457,155.451
C06118=1073.378,334.688,403.161,175.036,30.463,155.452
C06119=1073.384,334.936,403.127,175.039,30.467,155.453
C06120=1073.391,335.184,403.092,175.043,30.472,155.454
C06121=1073.397,335.431,403.058,175.046,30.477,155.454
C06122=1073.403,335.679,403.024,175.050,30.482,155.455
C06123=1073.409,335.926,402.990,175.052,30.487,155.456
C06124=1073.416,336.173,402.955,175.056,30.492,155.457
C06125=1073.422,336.421,402.921,175.059,30.497,155.458
C06126=1073.428,336.669,402.886,175.063,30.502,155.459
C06127=1073.434,336.916,402.852,175.066,30.508,155.460
C06128=1073.440,337.164,402.818,175.069,30.513,155.461
C06129=1073.447,337.412,402.783,175.073,30.518,155.462
C06130=1073.453,337.659,402.749,175.076,30.523,155.463
C06131=1073.459,337.907,402.714,175.080,30.528,155.464
C06132=1073.465,338.154,402.680,175.082,30.532,155.465
C06133=1073.472,338.401,402.645,175.086,30.538,155.466
C06134=1073.477,338.649,402.610,175.089,30.543,155.467
C06135=1073.484,338.897,402.576,175.093,30.548,155.467
C06136=1073.490,339.144,402.541,175.096,30.553,155.468
C06137=1073.496,339.391,402.507,175.099,30.558,155.469
C06138=1073.502,339.640,402.472,175.103,30.563,155.470
C06139=1073.508,339.886,402.437,175.106,30.568,155.471
C06140=1073.515,340.134,402.402,175.110,30.574,155.472
C06141=1073.521,340.382,402.367,175.112,30.579,155.473
C06142=1073.526,340.629,402.333,175.116,30.584,155.474
C06143=1073.533,340.877,402.298,175.120,30.589,155.475
C06144=1073.540,341.125,402.263,175.123,30.594,155.476
C06145=1073.546,341.371,402.228,175.127,30.600,155.477
C06146=1073.552,341.620,402.193,175.129,30.604,155.478
C06147=1073.558,341.867,402.158,175.133,30.610,155.479
C06148=1073.564,342.114,402.124,175.136,30.615,155.480
C06149=1073.571,342.362,402.089,175.140,30.620,155.481
C06150=1073.577,342.609,402.053,175.144,30.625,155.482
C06151=1073.583,342.857,402.019,175.147,30.630,155.483
C06152=1073.590,343.104,401.984,175.150,30.636,155.484
C06153=1073.596,343.352,401.948,175.153,30.641,155.485
C06154=1073.602,343.600,401.914,175.157,30.646,155.486
C06155=1073.608,343.846,401.879,175.160,30.651,155.487
C06156=1073.614,344.063,401.848,175.163,30.656,155.488
C06157=1073.619,344.279,401.818,175.167,30.660,155.488
C06158=1073.625,344.496,401.786,175.169,30.665,155.489
C06159=1073.630,344.711,401.756,175.172,30.670,155.490
C06160=1073.635,344.929,401.726,175.176,30.674,155.491
C06161=1073.641,345.144,401.695,175.178,30.679,155.492
C06162=1073.647,345.361,401.664,175.182,30.684,155.493
C06163=1073.651,345.577,401.633,175.184,30.688,155.494
C06164=1073.658,345.825,401.598,175.188,30.694,155.495
C06165=1073.664,346.072,401.562,175.192,30.699,155.496
C06166=1073.671,346.320,401.527,175.195,30.704,155.497
C06167=1073.676,346.567,401.492,175.198,30.710,155.498
C06168=1073.683,346.814,401.457,175.201,30.715,155.499
C06169=1073.689,347.062,401.421,175.205,30.721,155.500
C06170=1073.696,347.309,401.386,175.208,30.726,155.501
C06171=1073.702,347.557,401.350,175.212,30.731,155.502
C06172=1073.709,347.804,401.315,175.216,30.737,155.503
C06173=1073.714,348.051,401.280,175.219,30.742,155.504
C06174=1073.721,348.298,401.245,175.223,30.748,155.505
C06175=1073.727,348.546,401.209,175.226,30.753,155.506
C06176=1073.733,348.794,401.173,175.230,30.759,155.507
C06177=1073.740,349.041,401.138,175.232,30.764,155.508
C06178=1073.746,349.289,401.102,175.236,30.769,155.509
C06179=1073.752,349.536,401.066,175.240,30.775,155.510
C06180=1073.758,349.783,401.031,175.243,30.780,155.511
C06181=1073.764,350.030,400.995,175.247,30.786,155.512
C06182=1073.770,350.278,400.960,175.250,30.791,155.513
C06183=1073.777,350.525,400.924,175.254,30.797,155.514
C06184=1073.783,350.772,400.888,175.258,30.802,155.515
C06185=1073.790,351.020,400.853,175.261,30.808,155.516
C06186=1073.796,351.267,400.817,175.265,30.813,155.517
C06187=1073.803,351.514,400.781,175.268,30.819,155.518
C06188=1073.809,351.762,400.746,175.272,30.824,155.519
C06189=1073.815,352.009,400.710,175.275,30.830,155.520
C06190=1073.822,352.257,400.673,175.279,30.835,155.521
C06191=1073.828,352.504,400.638,175.283,30.841,155.522
C06192=1073.835,352.752,400.602,175.286,30.847,155.524
C06193=1073.841,352.999,400.566,175.290,30.852,155.525
C06194=1073.847,353.246,400.530,175.293,30.857,155.526
C06195=1073.853,353.493,400.494,175.297,30.863,155.527
C06196=1073.859,353.741,400.458,175.301,30.869,155.528
C06197=1073.866,353.988,400.422,175.304,30.874,155.529
C06198=1073.872,354.236,400.386,175.308,30.880,155.530
C06199=1073.879,354.483,400.350,175.310,30.886,155.531
C06200=1073.885,354.730,400.314,175.314,30.891,155.532
C06201=1073.891,354.977,400.278,175.318,30.897,155.533
C06202=1073.897,355.224,400.241,175.321,30.903,155.534
C06203=1073.903,355.472,400.206,175.325,30.909,155.535
C06204=1073.910,355.719,400.169,175.328,30.914,155.536
C06205=1073.916,355.966,400.133,175.333,30.920,155.538
C06206=1073.922,356.214,400.097,175.336,30.926,155.539
C06207=1073.928,356.461,400.061,175.340,30.932,155.540
C06208=1073.935,356.708,400.024,175.344,30.937,155.541
C06209=1073.941,356.956,399.988,175.347,30.943,155.542
C06210=1073.948,357.203,399.952,175.351,30.948,155.543
C06211=1073.954,357.450,399.915,175.354,30.954,155.544
C06212=1073.960,357.668,399.884,175.357,30.959,155.545
C06213=1073.965,357.886,399.851,175.361,30.965,155.546
C06214=1073.971,358.104,399.819,175.363,30.969,155.547
C06215=1073.977,358.322,399.788,175.367,30.975,155.548
C06216=1073.983,358.541,399.755,175.371,30.980,155.549
C06217=1073.988,358.759,399.723,175.373,30.985,155.550
C06218=1073.994,358.976,399.691,175.377,30.990,155.551
C06219=1073.999,359.195,399.658,175.380,30.995,155.552
C06220=1074.006,359.442,399.622,175.383,31.001,155.553
C06221=1074.012,359.689,399.586,175.387,31.007,155.554
C06222=1074.018,359.936,399.549,175.390,31.013,155.556
C06223=1074.025,360.183,399.513,175.395,31.019,155.557
C06224=1074.032,360.431,399.476,175.399,31.025,155.558
C06225=1074.038,360.678,399.439,175.402,31.031,155.559
C06226=1074.044,360.925,399.403,175.406,31.037,155.560
C06227=1074.050,361.172,399.366,175.409,31.042,155.561
C06228=1074.057,361.419,399.328,175.413,31.048,155.563
C06229=1074.064,361.666,399.292,175.417,31.054,155.564
C06230=1074.070,361.914,399.256,175.420,31.060,155.565
C06231=1074.076,362.161,399.219,175.424,31.066,155.566
C06232=1074.083,362.408,399.182,175.427,31.072,155.567
C06233=1074.089,362.656,399.145,175.431,31.078,155.568
C06234=1074.095,362.902,399.108,175.436,31.084,155.569
C06235=1074.102,363.149,399.072,175.439,31.090,155.571
C06236=1074.109,363.397,399.035,175.443,31.096,155.572
C06237=1074.115,363.644,398.997,175.446,31.102,155.573
C06238=1074.121,363.891,398.961,175.450,31.108,155.574
C06239=1074.128,364.139,398.924,175.454,31.114,155.575
C06240=1074.135,364.385,398.887,175.457,31.120,155.577
C06241=1074.140,364.632,398.850,175.461,31.126,155.578
C06242=1074.147,364.880,398.813,175.465,31.133,155.579
C06243=1074.154,365.127,398.776,175.469,31.138,155.580
C06244=1074.160,365.375,398.738,175.473,31.145,155.581
C06245=1074.167,365.621,398.701,175.476,31.151,155.583
C06246=1074.172,365.868,398.664,175.480,31.157,155.584
C06247=1074.179,366.116,398.627,175.483,31.163,155.585
C06248=1074.186,366.362,398.589,175.487,31.170,155.586
C06249=1074.192,366.609,398.552,175.492,31.176,155.587
C06250=1074.199,366.856,398.515,175.495,31.182,155.589
C06251=1074.205,367.104,398.478,175.499,31.188,155.590
C06252=1074.211,367.350,398.441,175.503,31.195,155.591
C06253=1074.218,367.598,398.402,175.506,31.201,155.592
C06254=1074.224,367.845,398.366,175.511,31.207,155.594
C06255=1074.231,368.092,398.328,175.514,31.214,155.595
C06256=1074.237,368.339,398.291,175.518,31.220,155.596
C06257=1074.244,368.586,398.253,175.522,31.226,155.597
C06258=1074.250,368.833,398.216,175.525,31.232,155.599
C06259=1074.256,369.080,398.178,175.530,31.238,155.600
C06260=1074.263,369.327,398.141,175.533,31.245,155.601
C06261=1074.269,369.574,398.103,175.537,31.251,155.602
C06262=1074.276,369.821,398.066,175.541,31.258,155.604
C06263=1074.282,370.068,398.029,175.544,31.264,155.605
C06264=1074.288,370.316,397.990,175.549,31.270,155.606
C06265=1074.295,370.562,397.953,175.553,31.277,155.608
C06266=1074.302,370.810,397.915,175.556,31.283,155.609
C06267=1074.309,371.057,397.878,175.560,31.290,155.610
C06268=1074.315,371.324,397.836,175.564,31.297,155.612
C06269=1074.323,371.592,397.796,175.569,31.304,155.613
C06270=1074.329,371.859,397.755,175.573,31.310,155.614
C06271=1074.337,372.126,397.714,175.577,31.317,155.616
C06272=1074.344,372.373,397.676,175.581,31.324,155.617
C06273=1074.350,372.620,397.639,175.585,31.330,155.618
C06274=1074.357,372.867,397.600,175.589,31.337,155.620
C06275=1074.363,373.114,397.563,175.593,31.343,155.621
C06276=1074.370,373.361,397.525,175.596,31.350,155.622
C06277=1074.376,373.608,397.487,175.600,31.357,155.624
C06278=1074.383,373.855,397.449,175.605,31.363,155.625
C06279=1074.389,374.102,397.410,175.608,31.370,155.626
C06280=1074.396,374.348,397.373,175.612,31.376,155.628
C06281=1074.402,374.596,397.335,175.616,31.383,155.629
C06282=1074.409,374.843,397.296,175.620,31.390,155.630
C06283=1074.415,375.089,397.259,175.624,31.396,155.632
C06284=1074.422,375.337,397.220,175.628,31.403,155.633
C06285=1074.428,375.584,397.182,175.632,31.410,155.634
C06286=1074.434,375.831,397.144,175.636,31.417,155.636
C06287=1074.441,376.077,397.105,175.639,31.423,155.637
C06288=1074.448,376.324,397.068,175.644,31.430,155.638
C06289=1074.455,376.571,397.029,175.648,31.437,155.640
C06290=1074.461,376.818,396.991,175.651,31.444,155.641
C06291=1074.468,377.065,396.952,175.656,31.450,155.642
C06292=1074.474,377.312,396.914,175.660,31.457,155.644
C06293=1074.481,377.558,396.876,175.663,31.464,155.645
C06294=1074.487,377.806,396.837,175.668,31.471,155.647
C06295=1074.494,378.053,396.799,175.672,31.477,155.648
C06296=1074.501,378.300,396.760,175.675,31.484,155.649
C06297=1074.507,378.546,396.722,175.680,31.491,155.651
C06298=1074.513,378.793,396.683,175.684,31.498,155.652
C06299=1074.520,379.040,396.644,175.687,31.505,155.654
C06300=1074.527,379.287,396.607,175.692,31.512,155.655
C06301=1074.534,379.534,396.568,175.696,31.519,155.656
C06302=1074.540,379.780,396.529,175.700,31.526,155.658
C06303=1074.547,380.027,396.491,175.704,31.533,155.659
C06304=1074.554,380.274,396.452,175.708,31.540,155.661
C06305=1074.561,380.521,396.414,175.712,31.547,155.662
C06306=1074.567,380.768,396.375,175.716,31.553,155.664
C06307=1074.574,381.015,396.336,175.721,31.561,155.665
C06308=1074.580,381.231,396.302,175.724,31.567,155.666
C06309=1074.586,381.446,396.268,175.727,31.573,155.667
C06310=1074.592,381.662,396.234,175.731,31.579,155.669
C06311=1074.598,381.879,396.200,175.734,31.585,155.670
C06312=1074.603,382.094,396.166,175.738,31.591,155.671
C06313=1074.609,382.311,396.132,175.742,31.597,155.673
C06314=1074.615,382.527,396.098,175.746,31.604,155.674
C06315=1074.621,382.743,396.064,175.749,31.610,155.675
C06316=1074.627,382.989,396.024,175.753,31.617,155.677
C06317=1074.633,383.236,395.986,175.758,31.625,155.678
C06318=1074.640,383.483,395.947,175.761,31.632,155.680
C06319=1074.647,383.730,395.908,175.765,31.639,155.681
C06320=1074.653,383.977,395.869,175.770,31.646,155.683
C06321=1074.660,384.224,395.830,175.773,31.653,155.684
C06322=1074.667,384.470,395.790,175.778,31.661,155.686
C06323=1074.673,384.717,395.751,175.782,31.668,155.687
C06324=1074.679,384.958,395.713,175.786,31.675,155.689
C06325=1074.686,385.199,395.674,175.790,31.682,155.690
C06326=1074.693,385.439,395.636,175.794,31.690,155.692
C06327=1074.700,385.681,395.597,175.798,31.697,155.693
C06328=1074.706,385.922,395.559,175.802,31.704,155.695
C06329=1074.713,386.162,395.520,175.807,31.711,155.696
C06330=1074.719,386.403,395.482,175.811,31.718,155.698
C06331=1074.726,386.645,395.444,175.814,31.725,155.699
C06332=1074.733,386.891,395.405,175.819,31.733,155.701
C06333=1074.739,387.138,395.365,175.823,31.740,155.702
C06334=1074.746,387.384,395.326,175.827,31.748,155.704
C06335=1074.752,387.631,395.286,175.832,31.755,155.705
C06336=1074.759,387.878,395.247,175.836,31.762,155.707
C06337=1074.766,388.124,395.208,175.840,31.770,155.708
C06338=1074.773,388.372,395.167,175.844,31.777,155.710
C06339=1074.780,388.618,395.128,175.849,31.785,155.712
C06340=1074.787,388.865,395.089,175.853,31.793,155.713
C06341=1074.794,389.111,395.049,175.857,31.800,155.715
C06342=1074.800,389.358,395.010,175.861,31.808,155.716
C06343=1074.807,389.605,394.969,175.866,31.815,155.718
C06344=1074.814,389.851,394.930,175.870,31.823,155.720
C06345=1074.822,390.098,394.890,175.874,31.831,155.721
C06346=1074.828,390.344,394.850,175.879,31.838,155.723
C06347=1074.835,390.592,394.811,175.883,31.846,155.724
C06348=1074.842,390.838,394.771,175.887,31.853,155.726
C06349=1074.849,391.084,394.731,175.892,31.861,155.728
C06350=1074.855,391.331,394.691,175.896,31.869,155.729
C06351=1074.863,391.578,394.651,175.901,31.877,155.731
C06352=1074.869,391.824,394.611,175.905,31.885,155.732
C06353=1074.876,392.071,394.571,175.909,31.893,155.734
C06354=1074.883,392.317,394.531,175.914,31.900,155.736
C06355=1074.890,392.564,394.491,175.917,31.908,155.737
C06356=1074.896,392.811,394.451,175.922,31.916,155.739
C06357=1074.903,393.057,394.411,175.927,31.924,155.741
C06358=1074.910,393.304,394.371,175.931,31.932,155.742
C06359=1074.917,393.551,394.330,175.935,31.940,155.744
C06360=1074.924,393.797,394.291,175.940,31.948,155.746
C06361=1074.931,394.044,394.250,175.944,31.956,155.748
C06362=1074.937,394.290,394.209,175.949,31.964,155.749
C06363=1074.944,394.537,394.169,175.953,31.972,155.751
C06364=1074.952,394.783,394.129,175.957,31.979,155.753
C06365=1074.958,395.030,394.089,175.962,31.987,155.754
C06366=1074.965,395.276,394.048,175.967,31.996,155.756
C06367=1074.972,395.523,394.008,175.970,32.004,155.758
C06368=1074.979,395.770,393.967,175.975,32.012,155.759
C06369=1074.985,396.016,393.927,175.980,32.020,155.761
C06370=1074.993,396.263,393.887,175.985,32.028,155.763
C06371=1074.999,396.509,393.846,175.988,32.036,155.765
C06372=1075.007,396.756,393.805,175.993,32.044,155.766
C06373=1075.013,397.003,393.765,175.998,32.053,155.768
C06374=1075.020,397.249,393.724,176.002,32.061,155.770
C06375=1075.027,397.496,393.684,176.006,32.069,155.772
C06376=1075.034,397.742,393.642,176.011,32.078,155.774
C06377=1075.040,397.989,393.602,176.016,32.086,155.775
C06378=1075.048,398.235,393.562,176.020,32.094,155.777
C06379=1075.056,398.482,393.520,176.025,32.102,155.779
C06380=1075.062,398.732,393.479,176.029,32.111,155.781
C06381=1075.069,398.983,393.437,176.034,32.119,155.783
C06382=1075.076,399.232,393.396,176.039,32.128,155.784
C06383=1075.083,399.483,393.354,176.044,32.137,155.786
C06384=1075.090,399.730,393.314,176.047,32.145,155.788
C06385=1075.097,399.976,393.273,176.052,32.154,155.790
C06386=1075.104,400.223,393.232,176.057,32.162,155.792
C06387=1075.111,400.469,393.190,176.062,32.170,155.794
C06388=1075.118,400.715,393.149,176.067,32.179,155.796
C06389=1075.125,400.962,393.108,176.070,32.188,155.797
C06390=1075.132,401.209,393.068,176.075,32.196,155.799
C06391=1075.139,401.456,393.026,176.080,32.205,155.801
C06392=1075.145,401.702,392.985,176.085,32.214,155.803
C06393=1075.153,401.948,392.944,176.090,32.222,155.805
C06394=1075.160,402.195,392.903,176.095,32.231,155.807
C06395=1075.167,402.442,392.861,176.098,32.239,155.809
C06396=1075.174,402.688,392.820,176.103,32.248,155.810
C06397=1075.181,402.934,392.779,176.108,32.257,155.812
C06398=1075.188,403.180,392.737,176.113,32.266,155.814
C06399=1075.195,403.427,392.695,176.118,32.274,155.816
C06400=1075.203,403.674,392.654,176.122,32.283,155.818
C06401=1075.210,403.920,392.613,176.127,32.292,155.820
C06402=1075.216,404.166,392.572,176.132,32.301,155.822
C06403=1075.223,404.412,392.530,176.137,32.310,155.824
C06404=1075.231,404.659,392.488,176.142,32.319,155.826
C06405=1075.237,404.906,392.447,176.147,32.328,155.828
C06406=1075.245,405.152,392.405,176.150,32.337,155.830
C06407=1075.252,405.398,392.363,176.155,32.346,155.832
C06408=1075.259,405.645,392.322,176.160,32.355,155.834
C06409=1075.266,405.891,392.280,176.165,32.364,155.836
C06410=1075.273,406.138,392.238,176.170,32.373,155.838
C06411=1075.280,406.384,392.196,176.175,32.382,155.840
C06412=1075.287,406.630,392.155,176.180,32.391,155.842
C06413=1075.294,406.876,392.112,176.184,32.400,155.844
C06414=1075.301,407.123,392.071,176.189,32.410,155.846
C06415=1075.308,407.369,392.029,176.194,32.419,155.848
C06416=1075.315,407.616,391.986,176.199,32.428,155.850
C06417=1075.322,407.862,391.945,176.204,32.437,155.852
C06418=1075.329,408.108,391.902,176.209,32.447,155.854
C06419=1075.337,408.354,391.860,176.214,32.456,155.856
C06420=1075.343,408.601,391.819,176.219,32.466,155.858
C06421=1075.351,408.847,391.777,176.224,32.474,155.860
C06422=1075.358,409.094,391.734,176.228,32.484,155.862
C06423=1075.365,409.341,391.691,176.234,32.494,155.864
C06424=1075.373,409.587,391.649,176.239,32.503,155.866
C06425=1075.380,409.833,391.607,176.244,32.513,155.869
C06426=1075.386,410.080,391.565,176.249,32.522,155.871
C06427=1075.394,410.326,391.523,176.254,32.531,155.873
C06428=1075.401,410.572,391.480,176.259,32.541,155.875
C06429=1075.407,410.818,391.438,176.264,32.551,155.877
C06430=1075.415,411.064,391.396,176.269,32.560,155.879
C06431=1075.423,411.311,391.353,176.274,32.570,155.881
C06432=1075.430,411.557,391.310,176.280,32.579,155.883
C06433=1075.437,411.803,391.268,176.284,32.589,155.886
C06434=1075.444,412.049,391.225,176.289,32.599,155.888
C06435=1075.451,412.295,391.183,176.294,32.609,155.890
C06436=1075.460,412.549,391.139,176.299,32.618,155.892
C06437=1075.467,412.803,391.095,176.305,32.629,155.894
C06438=1075.475,413.056,391.051,176.310,32.639,155.897
C06439=1075.482,413.310,391.007,176.316,32.649,155.899
C06440=1075.489,413.556,390.964,176.321,32.659,155.901
C06441=1075.496,413.802,390.922,176.326,32.668,155.903
C06442=1075.504,414.048,390.879,176.331,32.678,155.905
C06443=1075.511,414.295,390.836,176.337,32.688,155.908
C06444=1075.518,414.541,390.794,176.342,32.698,155.910
C06445=1075.526,414.787,390.751,176.347,32.708,155.912
C06446=1075.533,415.033,390.708,176.352,32.718,155.914
C06447=1075.541,415.280,390.664,176.358,32.728,155.917
C06448=1075.548,415.525,390.621,176.363,32.739,155.919
C06449=1075.555,415.772,390.579,176.368,32.748,155.921
C06450=1075.563,416.018,390.535,176.374,32.759,155.924
C06451=1075.570,416.264,390.492,176.379,32.769,155.926
C06452=1075.577,416.511,390.449,176.384,32.779,155.928
C06453=1075.585,416.756,390.406,176.389,32.789,155.930
C06454=1075.592,417.003,390.362,176.395,32.800,155.933
C06455=1075.600,417.248,390.319,176.400,32.810,155.935
C06456=1075.606,417.495,390.276,176.406,32.821,155.938
C06457=1075.614,417.741,390.233,176.411,32.831,155.940
C06458=1075.621,417.987,390.189,176.416,32.841,155.942
C06459=1075.629,418.233,390.146,176.422,32.852,155.945
C06460=1075.636,418.479,390.102,176.427,32.862,155.947
C06461=1075.644,418.725,390.059,176.433,32.873,155.949
C06462=1075.652,418.971,390.015,176.438,32.883,155.952
C06463=1075.658,419.217,389.971,176.443,32.894,155.954
C06464=1075.666,419.464,389.928,176.449,32.904,155.957
C06465=1075.673,419.709,389.884,176.454,32.915,155.959
C06466=1075.681,419.955,389.840,176.460,32.926,155.961
C06467=1075.689,420.201,389.796,176.466,32.936,155.964
C06468=1075.696,420.447,389.753,176.472,32.947,155.966
C06469=1075.704,420.693,389.710,176.477,32.958,155.969
C06470=1075.712,420.940,389.666,176.483,32.969,155.971
C06471=1075.719,421.185,389.622,176.488,32.979,155.974
C06472=1075.726,421.432,389.578,176.494,32.990,155.976
C06473=1075.734,421.678,389.534,176.499,33.001,155.979
C06474=1075.742,421.924,389.490,176.505,33.012,155.981
C06475=1075.748,422.170,389.446,176.510,33.023,155.984
C06476=1075.756,422.415,389.402,176.516,33.034,155.986
C06477=1075.764,422.662,389.358,176.522,33.045,155.989
C06478=1075.771,422.907,389.313,176.528,33.056,155.991
C06479=1075.779,423.153,389.269,176.534,33.068,155.994
C06480=1075.787,423.399,389.225,176.539,33.078,155.996
C06481=1075.794,423.645,389.181,176.545,33.090,155.999
C06482=1075.802,423.891,389.136,176.550,33.101,156.002
C06483=1075.809,424.137,389.092,176.556,33.112,156.004
C06484=1075.817,424.383,389.048,176.563,33.124,156.007
C06485=1075.824,424.629,389.003,176.568,33.135,156.009
C06486=1075.832,424.875,388.959,176.574,33.146,156.012
C06487=1075.840,425.120,388.914,176.580,33.158,156.015
C06488=1075.847,425.367,388.870,176.585,33.169,156.017
C06489=1075.855,425.613,388.826,176.591,33.180,156.020
C06490=1075.863,425.859,388.781,176.598,33.192,156.023
C06491=1075.870,426.104,388.737,176.603,33.203,156.025
C06492=1075.879,426.375,388.687,176.610,33.216,156.028
C06493=1075.887,426.646,388.637,176.616,33.229,156.031
C06494=1075.896,426.918,388.589,176.623,33.241,156.034
C06495=1075.904,427.189,388.539,176.630,33.254,156.037
C06496=1075.913,427.435,388.495,176.636,33.266,156.040
C06497=1075.920,427.681,388.449,176.641,33.278,156.043
C06498=1075.928,427.926,388.405,176.648,33.289,156.045
C06499=1075.936,428.172,388.360,176.654,33.302,156.048
C06500=1075.943,428.418,388.314,176.660,33.313,156.051
C06501=1075.951,428.664,388.269,176.666,33.325,156.054
C06502=1075.959,428.910,388.225,176.672,33.337,156.056
C06503=1075.966,429.155,388.179,176.678,33.349,156.059
C06504=1075.974,429.401,388.134,176.684,33.361,156.062
C06505=1075.982,429.646,388.089,176.691,33.373,156.065
C06506=1075.989,429.892,388.044,176.697,33.385,156.068
C06507=1075.998,430.138,387.998,176.703,33.397,156.071
C06508=1076.005,430.384,387.953,176.710,33.410,156.073
C06509=1076.013,430.630,387.908,176.716,33.422,156.076
C06510=1076.021,430.875,387.863,176.721,33.434,156.079
C06511=1076.029,431.120,387.817,176.728,33.446,156.082
C06512=1076.037,431.367,387.771,176.734,33.459,156.085
C06513=1076.044,431.613,387.726,176.740,33.471,156.088
C06514=1076.053,431.858,387.681,176.747,33.483,156.091
C06515=1076.061,432.104,387.635,176.753,33.496,156.094
C06516=1076.068,432.349,387.589,176.759,33.508,156.097
C06517=1076.076,432.595,387.544,176.766,33.521,156.100
C06518=1076.084,432.840,387.498,176.772,33.534,156.103
C06519=1076.092,433.086,387.452,176.779,33.546,156.106
C06520=1076.100,433.332,387.406,176.785,33.559,156.109
C06521=1076.107,433.577,387.361,176.791,33.571,156.112
C06522=1076.116,433.823,387.314,176.798,33.584,156.115
C06523=1076.123,434.068,387.268,176.804,33.597,156.118
C06524=1076.131,434.314,387.223,176.811,33.610,156.121
C06525=1076.139,434.560,387.177,176.818,33.623,156.124
C06526=1076.147,434.805,387.130,176.825,33.635,156.127
C06527=1076.156,435.051,387.084,176.831,33.649,156.130
C06528=1076.163,435.296,387.039,176.838,33.661,156.133
C06529=1076.171,435.542,386.991,176.844,33.675,156.136
C06530=1076.179,435.787,386.946,176.851,33.688,156.139
C06531=1076.187,436.033,386.899,176.857,33.700,156.142
C06532=1076.195,436.278,386.853,176.864,33.714,156.146
C06533=1076.203,436.524,386.807,176.871,33.727,156.149
C06534=1076.211,436.769,386.760,176.878,33.740,156.152
C06535=1076.220,437.015,386.714,176.884,33.753,156.155
C06536=1076.227,437.260,386.668,176.891,33.767,156.158
C06537=1076.236,437.505,386.621,176.898,33.780,156.162
C06538=1076.245,437.751,386.574,176.905,33.793,156.165
C06539=1076.251,437.996,386.528,176.912,33.807,156.168
C06540=1076.260,438.242,386.481,176.918,33.821,156.171
C06541=1076.269,438.487,386.435,176.926,33.834,156.174
C06542=1076.276,438.732,386.388,176.932,33.847,156.178
C06543=1076.285,438.978,386.342,176.939,33.861,156.181
C06544=1076.294,439.223,386.295,176.947,33.875,156.184
C06545=1076.301,439.469,386.248,176.953,33.888,156.188
C06546=1076.309,439.714,386.201,176.960,33.903,156.191
C06547=1076.317,439.959,386.153,176.968,33.916,156.194
C06548=1076.326,440.223,386.103,176.974,33.931,156.198
C06549=1076.335,440.488,386.052,176.982,33.946,156.202
C06550=1076.344,440.752,386.002,176.990,33.961,156.205
C06551=1076.353,441.017,385.951,176.998,33.976,156.209
C06552=1076.362,441.261,385.904,177.005,33.991,156.213
C06553=1076.370,441.507,385.856,177.012,34.005,156.216
C06554=1076.378,441.752,385.809,177.020,34.019,156.219
C06555=1076.386,441.998,385.761,177.026,34.033,156.223
C06556=1076.395,442.243,385.714,177.034,34.048,156.226
C06557=1076.403,442.489,385.667,177.041,34.062,156.230
C06558=1076.412,442.734,385.619,177.049,34.076,156.233
C06559=1076.420,442.979,385.571,177.056,34.090,156.237
C06560=1076.428,443.224,385.524,177.063,34.105,156.240
C06561=1076.436,443.469,385.476,177.070,34.120,156.244
C06562=1076.445,443.714,385.429,177.078,34.134,156.248
C06563=1076.453,443.960,385.381,177.085,34.149,156.251
C06564=1076.462,444.204,385.333,177.093,34.163,156.255
C06565=1076.470,444.450,385.285,177.101,34.178,156.258
C06566=1076.478,444.695,385.237,177.108,34.193,156.262
C06567=1076.487,444.940,385.190,177.115,34.208,156.266
C06568=1076.495,445.185,385.142,177.123,34.223,156.269
C06569=1076.504,445.430,385.094,177.130,34.238,156.273
C06570=1076.512,445.675,385.046,177.138,34.253,156.277
C06571=1076.521,445.921,384.998,177.146,34.268,156.281
C06572=1076.530,446.166,384.949,177.153,34.283,156.284
C06573=1076.538,446.411,384.901,177.161,34.298,156.288
C06574=1076.546,446.656,384.853,177.169,34.313,156.292
C06575=1076.556,446.901,384.805,177.176,34.328,156.296
C06576=1076.564,447.146,384.757,177.183,34.344,156.299
C06577=1076.572,447.391,384.708,177.190,34.359,156.303
C06578=1076.580,447.636,384.660,177.197,34.374,156.307
C06579=1076.590,447.881,384.611,177.203,34.389,156.311
C06580=1076.598,448.126,384.563,177.209,34.404,156.315
C06581=1076.606,448.371,384.515,177.215,34.419,156.318
C06582=1076.616,448.615,384.466,177.221,34.434,156.322
C06583=1076.624,448.859,384.418,177.226,34.450,156.326
C06584=1076.635,449.104,384.370,177.231,34.464,156.330
C06585=1076.646,449.349,384.324,177.236,34.478,156.333
C06586=1076.660,449.595,384.277,177.241,34.491,156.337
C06587=1076.674,449.841,384.233,177.246,34.504,156.340
C06588=1076.315,449.837,383.998,177.225,34.660,156.381
C06589=1076.301,449.590,384.043,177.221,34.648,156.378
C06590=1076.287,449.345,384.089,177.216,34.634,156.375
C06591=1076.275,449.100,384.137,177.210,34.621,156.371
C06592=1076.265,448.856,384.183,177.204,34.606,156.368
C06593=1076.256,448.610,384.232,177.199,34.592,156.364
C06594=1076.247,448.366,384.280,177.193,34.576,156.360
C06595=1076.238,448.121,384.329,177.188,34.561,156.356
C06596=1076.230,447.877,384.378,177.181,34.546,156.352
C06597=1076.221,447.632,384.426,177.174,34.531,156.348
C06598=1076.212,447.387,384.474,177.167,34.516,156.345
C06599=1076.203,447.142,384.523,177.161,34.500,156.341
C06600=1076.195,446.897,384.572,177.153,34.485,156.337
C06601=1076.186,446.652,384.619,177.146,34.470,156.333
C06602=1076.178,446.407,384.667,177.138,34.455,156.329
C06603=1076.169,446.162,384.716,177.130,34.440,156.326
C06604=1076.161,445.917,384.764,177.123,34.425,156.322
C06605=1076.152,445.671,384.812,177.115,34.410,156.318
C06606=1076.143,445.427,384.861,177.107,34.395,156.315
C06607=1076.135,445.181,384.909,177.100,34.380,156.311
C06608=1076.127,444.936,384.957,177.092,34.365,156.307
C06609=1076.118,444.691,385.004,177.084,34.350,156.303
C06610=1076.110,444.446,385.052,177.077,34.335,156.300
C06611=1076.102,444.201,385.100,177.069,34.321,156.296
C06612=1076.092,443.955,385.148,177.061,34.305,156.292
C06613=1076.084,443.710,385.196,177.054,34.291,156.289
C06614=1076.075,443.465,385.244,177.046,34.276,156.285
C06615=1076.067,443.220,385.292,177.039,34.262,156.282
C06616=1076.058,442.975,385.339,177.031,34.248,156.278
C06617=1076.050,442.730,385.387,177.024,34.233,156.275
C06618=1076.042,442.484,385.434,177.016,34.219,156.271
C06619=1076.034,442.239,385.482,177.009,34.204,156.268
C06620=1076.025,441.994,385.529,177.002,34.190,156.264
C06621=1076.017,441.749,385.577,176.995,34.176,156.261
C06622=1076.008,441.504,385.624,176.987,34.162,156.257
C06623=1076.000,441.258,385.672,176.980,34.148,156.254
C06624=1075.992,441.014,385.719,176.972,34.133,156.250
C06625=1075.983,440.766,385.766,176.965,34.119,156.247
C06626=1075.975,440.519,385.814,176.958,34.105,156.243
C06627=1075.967,440.273,385.861,176.951,34.091,156.240
C06628=1075.958,440.025,385.908,176.943,34.077,156.237
C06629=1075.951,439.780,385.956,176.936,34.063,156.233
C06630=1075.942,439.535,386.003,176.930,34.050,156.230
C06631=1075.934,439.289,386.050,176.922,34.036,156.226
C06632=1075.926,439.044,386.097,176.915,34.022,156.223
C06633=1075.917,438.799,386.144,176.908,34.009,156.220
C06634=1075.909,438.553,386.190,176.901,33.995,156.217
C06635=1075.900,438.308,386.237,176.894,33.981,156.213
C06636=1075.892,438.063,386.283,176.887,33.968,156.210
C06637=1075.885,437.817,386.331,176.881,33.955,156.207
C06638=1075.876,437.571,386.377,176.873,33.941,156.203
C06639=1075.868,437.327,386.424,176.866,33.928,156.200
C06640=1075.860,437.081,386.470,176.860,33.915,156.197
C06641=1075.851,436.835,386.516,176.853,33.901,156.194
C06642=1075.843,436.590,386.563,176.846,33.888,156.191
C06643=1075.835,436.345,386.610,176.839,33.875,156.188
C06644=1075.827,436.099,386.655,176.832,33.862,156.184
C06645=1075.819,435.853,386.703,176.826,33.849,156.181
C06646=1075.811,435.607,386.749,176.819,33.836,156.178
C06647=1075.803,435.362,386.795,176.813,33.822,156.175
C06648=1075.796,435.117,386.841,176.805,33.810,156.172
C06649=1075.787,434.872,386.887,176.798,33.796,156.169
C06650=1075.779,434.626,386.933,176.792,33.784,156.166
C06651=1075.771,434.381,386.980,176.785,33.771,156.163
C06652=1075.763,434.135,387.025,176.779,33.758,156.159
C06653=1075.755,433.889,387.071,176.772,33.745,156.156
C06654=1075.747,433.644,387.117,176.766,33.732,156.153
C06655=1075.739,433.399,387.163,176.759,33.720,156.150
C06656=1075.731,433.153,387.209,176.753,33.707,156.147
C06657=1075.724,432.907,387.255,176.746,33.694,156.144
C06658=1075.715,432.661,387.301,176.740,33.682,156.141
C06659=1075.708,432.416,387.347,176.733,33.669,156.138
C06660=1075.700,432.170,387.392,176.727,33.657,156.135
C06661=1075.692,431.925,387.438,176.720,33.644,156.132
C06662=1075.684,431.679,387.484,176.714,33.632,156.130
C06663=1075.677,431.433,387.530,176.707,33.619,156.127
C06664=1075.668,431.188,387.575,176.701,33.607,156.124
C06665=1075.660,430.942,387.621,176.695,33.595,156.121
C06666=1075.653,430.696,387.666,176.688,33.583,156.118
C06667=1075.645,430.450,387.711,176.682,33.570,156.115
C06668=1075.637,430.205,387.756,176.675,33.558,156.112
C06669=1075.628,429.959,387.802,176.669,33.546,156.109
C06670=1075.621,429.713,387.847,176.664,33.534,156.106
C06671=1075.613,429.468,387.893,176.657,33.522,156.104
C06672=1075.605,429.222,387.937,176.651,33.510,156.101
C06673=1075.598,428.977,387.983,176.645,33.498,156.098
C06674=1075.590,428.730,388.028,176.638,33.486,156.095
C06675=1075.583,428.485,388.073,176.632,33.474,156.092
C06676=1075.574,428.239,388.118,176.626,33.462,156.090
C06677=1075.566,427.993,388.164,176.620,33.450,156.087
C06678=1075.559,427.747,388.209,176.614,33.438,156.084
C06679=1075.551,427.501,388.253,176.607,33.427,156.081
C06680=1075.544,427.255,388.298,176.601,33.415,156.079
C06681=1075.534,426.983,388.348,176.595,33.402,156.076
C06682=1075.526,426.711,388.398,176.588,33.390,156.073
C06683=1075.517,426.437,388.448,176.581,33.377,156.070
C06684=1075.509,426.164,388.496,176.575,33.364,156.067
C06685=1075.501,425.919,388.542,176.569,33.352,156.064
C06686=1075.493,425.673,388.586,176.563,33.341,156.061
C06687=1075.485,425.427,388.631,176.557,33.329,156.059
C06688=1075.478,425.181,388.676,176.551,33.318,156.056
C06689=1075.470,424.936,388.720,176.546,33.307,156.053
C06690=1075.463,424.689,388.764,176.539,33.295,156.051
C06691=1075.455,424.443,388.809,176.533,33.284,156.048
C06692=1075.447,424.197,388.853,176.528,33.273,156.045
C06693=1075.440,423.952,388.898,176.522,33.262,156.043
C06694=1075.432,423.706,388.942,176.515,33.250,156.040
C06695=1075.425,423.460,388.986,176.510,33.239,156.038
C06696=1075.417,423.214,389.030,176.504,33.228,156.035
C06697=1075.409,422.968,389.075,176.499,33.217,156.032
C06698=1075.402,422.722,389.119,176.492,33.205,156.030
C06699=1075.394,422.476,389.163,176.486,33.195,156.027
C06700=1075.387,422.230,389.208,176.481,33.183,156.025
C06701=1075.379,421.984,389.251,176.475,33.172,156.022
C06702=1075.372,421.739,389.295,176.470,33.162,156.020
C06703=1075.365,421.492,389.340,176.464,33.151,156.017
C06704=1075.357,421.246,389.383,176.458,33.140,156.015
C06705=1075.349,421.000,389.428,176.452,33.129,156.012
C06706=1075.342,420.755,389.471,176.447,33.118,156.010
C06707=1075.334,420.508,389.515,176.441,33.107,156.007
C06708=1075.326,420.262,389.559,176.436,33.097,156.005
C06709=1075.319,420.017,389.602,176.430,33.086,156.003
C06710=1075.312,419.770,389.646,176.424,33.076,156.000
C06711=1075.304,419.524,389.690,176.418,33.065,155.998
C06712=1075.296,419.279,389.734,176.413,33.054,155.995
C06713=1075.289,419.032,389.778,176.408,33.044,155.993
C06714=1075.281,418.786,389.821,176.402,33.033,155.990
C06715=1075.274,418.540,389.864,176.397,33.023,155.988
C06716=1075.266,418.294,389.908,176.391,33.012,155.986
C06717=1075.259,418.048,389.951,176.386,33.002,155.983
C06718=1075.251,417.802,389.995,176.381,32.991,155.981
C06719=1075.244,417.556,390.038,176.374,32.981,155.978
C06720=1075.236,417.310,390.082,176.369,32.971,155.976
C06721=1075.229,417.064,390.124,176.363,32.960,155.974
C06722=1075.222,416.817,390.168,176.358,32.950,155.971
C06723=1075.215,416.571,390.212,176.353,32.940,155.969
C06724=1075.207,416.325,390.255,176.347,32.930,155.967
C06725=1075.200,416.079,390.299,176.342,32.919,155.964
C06726=1075.193,415.832,390.342,176.337,32.909,155.962
C06727=1075.186,415.587,390.385,176.332,32.899,155.960
C06728=1075.178,415.341,390.428,176.326,32.889,155.958
C06729=1075.170,415.094,390.470,176.321,32.878,155.955
C06730=1075.163,414.849,390.514,176.316,32.868,155.953
C06731=1075.156,414.602,390.557,176.310,32.859,155.951
C06732=1075.148,414.356,390.600,176.305,32.849,155.949
C06733=1075.141,414.109,390.643,176.300,32.839,155.946
C06734=1075.133,413.864,390.685,176.295,32.829,155.944
C06735=1075.126,413.617,390.728,176.289,32.819,155.942
C06736=1075.119,413.370,390.771,176.284,32.809,155.940
C06737=1075.111,413.116,390.816,176.279,32.799,155.937
C06738=1075.103,412.861,390.860,176.273,32.789,155.935
C06739=1075.095,412.606,390.904,176.268,32.779,155.933
C06740=1075.088,412.351,390.947,176.263,32.769,155.931
C06741=1075.081,412.105,390.991,176.258,32.759,155.928
C06742=1075.074,411.859,391.033,176.252,32.749,155.926
C06743=1075.066,411.612,391.075,176.247,32.739,155.924
C06744=1075.059,411.366,391.118,176.242,32.730,155.922
C06745=1075.052,411.119,391.161,176.237,32.720,155.920
C06746=1075.044,410.873,391.202,176.232,32.710,155.918
C06747=1075.037,410.627,391.245,176.227,32.701,155.915
C06748=1075.030,410.380,391.288,176.222,32.692,155.913
C06749=1075.022,410.134,391.330,176.216,32.682,155.911
C06750=1075.015,409.888,391.372,176.211,32.672,155.909
C06751=1075.009,409.642,391.415,176.206,32.663,155.907
C06752=1075.001,409.396,391.457,176.201,32.654,155.905
C06753=1074.994,409.149,391.499,176.196,32.644,155.903
C06754=1074.987,408.903,391.542,176.191,32.635,155.901
C06755=1074.980,408.657,391.584,176.186,32.625,155.899
C06756=1074.973,408.411,391.626,176.181,32.616,155.897
C06757=1074.965,408.164,391.668,176.176,32.607,155.894
C06758=1074.958,407.917,391.711,176.171,32.597,155.892
C06759=1074.951,407.671,391.753,176.166,32.588,155.890
C06760=1074.944,407.425,391.795,176.161,32.579,155.888
C06761=1074.937,407.178,391.837,176.156,32.570,155.886
C06762=1074.930,406.932,391.879,176.151,32.560,155.884
C06763=1074.923,406.685,391.921,176.146,32.551,155.882
C06764=1074.915,406.439,391.963,176.142,32.542,155.880
C06765=1074.909,406.193,392.005,176.137,32.533,155.878
C06766=1074.902,405.947,392.046,176.132,32.524,155.876
C06767=1074.894,405.701,392.088,176.127,32.515,155.874
C06768=1074.888,405.454,392.130,176.122,32.506,155.872
C06769=1074.880,405.208,392.171,176.117,32.497,155.870
C06770=1074.874,404.961,392.214,176.112,32.487,155.868
C06771=1074.866,404.715,392.255,176.107,32.478,155.866
C06772=1074.859,404.469,392.297,176.102,32.470,155.864
C06773=1074.852,404.222,392.339,176.098,32.461,155.862
C06774=1074.845,403.975,392.380,176.094,32.452,155.860
C06775=1074.838,403.729,392.421,176.089,32.443,155.858
C06776=1074.831,403.483,392.463,176.084,32.435,155.857
C06777=1074.824,403.236,392.504,176.079,32.426,155.855
C06778=1074.817,402.990,392.546,176.074,32.417,155.853
C06779=1074.809,402.743,392.587,176.069,32.408,155.851
C06780=1074.802,402.497,392.628,176.064,32.399,155.849
C06781=1074.795,402.250,392.669,176.060,32.391,155.847
C06782=1074.788,402.004,392.710,176.056,32.382,155.845
C06783=1074.782,401.757,392.752,176.051,32.373,155.843
C06784=1074.774,401.511,392.793,176.046,32.365,155.841
C06785=1074.767,401.264,392.834,176.041,32.356,155.839
C06786=1074.760,401.018,392.875,176.036,32.347,155.838
C06787=1074.753,400.772,392.917,176.032,32.339,155.836
C06788=1074.746,400.525,392.958,176.027,32.330,155.834
C06789=1074.738,400.278,392.999,176.023,32.322,155.832
C06790=1074.732,400.033,393.040,176.018,32.313,155.830
C06791=1074.725,399.786,393.082,176.013,32.305,155.828
C06792=1074.718,399.538,393.122,176.009,32.297,155.827
C06793=1074.711,399.288,393.164,176.004,32.288,155.825
C06794=1074.704,399.036,393.206,175.999,32.279,155.823
C06795=1074.697,398.784,393.248,175.994,32.271,155.821
C06796=1074.689,398.532,393.290,175.990,32.262,155.819
C06797=1074.682,398.285,393.330,175.985,32.254,155.817
C06798=1074.676,398.039,393.371,175.981,32.245,155.816
C06799=1074.668,397.792,393.412,175.976,32.237,155.814
C06800=1074.662,397.546,393.452,175.971,32.229,155.812
C06801=1074.655,397.299,393.493,175.967,32.221,155.810
C06802=1074.648,397.052,393.534,175.963,32.212,155.808
C06803=1074.641,396.806,393.575,175.958,32.204,155.807
C06804=1074.634,396.559,393.615,175.953,32.196,155.805
C06805=1074.627,396.313,393.656,175.949,32.188,155.803
C06806=1074.620,396.066,393.696,175.944,32.180,155.801
C06807=1074.613,395.820,393.737,175.940,32.172,155.800
C06808=1074.606,395.573,393.778,175.935,32.163,155.798
C06809=1074.600,395.326,393.818,175.931,32.155,155.796
C06810=1074.592,395.080,393.859,175.926,32.147,155.794
C06811=1074.586,394.833,393.899,175.921,32.139,155.793
C06812=1074.579,394.587,393.939,175.918,32.131,155.791
C06813=1074.572,394.340,393.980,175.913,32.123,155.789
C06814=1074.565,394.094,394.020,175.908,32.115,155.788
C06815=1074.558,393.847,394.061,175.904,32.107,155.786
C06816=1074.551,393.601,394.100,175.899,32.099,155.784
C06817=1074.545,393.354,394.140,175.896,32.091,155.783
C06818=1074.538,393.107,394.181,175.891,32.083,155.781
C06819=1074.530,392.861,394.221,175.886,32.075,155.779
C06820=1074.524,392.615,394.261,175.882,32.068,155.777
C06821=1074.517,392.367,394.302,175.878,32.060,155.776
C06822=1074.510,392.121,394.341,175.873,32.052,155.774
C06823=1074.504,391.875,394.381,175.869,32.044,155.772
C06824=1074.497,391.628,394.422,175.864,32.036,155.771
C06825=1074.489,391.381,394.461,175.860,32.028,155.769
C06826=1074.483,391.135,394.502,175.856,32.020,155.767
C06827=1074.475,390.888,394.541,175.851,32.013,155.766
C06828=1074.469,390.641,394.582,175.847,32.005,155.764
C06829=1074.462,390.395,394.620,175.842,31.998,155.763
C06830=1074.456,390.148,394.661,175.838,31.990,155.761
C06831=1074.448,389.901,394.701,175.834,31.982,155.759
C06832=1074.441,389.655,394.740,175.829,31.975,155.758
C06833=1074.435,389.408,394.780,175.825,31.967,155.756
C06834=1074.428,389.162,394.819,175.821,31.959,155.755
C06835=1074.421,388.914,394.860,175.817,31.952,155.753
C06836=1074.414,388.668,394.899,175.812,31.945,155.752
C06837=1074.407,388.421,394.938,175.807,31.937,155.750
C06838=1074.400,388.175,394.978,175.804,31.929,155.748
C06839=1074.393,387.929,395.018,175.799,31.922,155.747
C06840=1074.387,387.682,395.057,175.795,31.914,155.745
C06841=1074.380,387.435,395.097,175.790,31.907,155.744
C06842=1074.373,387.188,395.136,175.787,31.900,155.742
C06843=1074.366,386.941,395.176,175.782,31.892,155.740
C06844=1074.359,386.694,395.215,175.778,31.885,155.739
C06845=1074.353,386.453,395.253,175.773,31.878,155.737
C06846=1074.347,386.211,395.292,175.770,31.870,155.736
C06847=1074.340,385.970,395.330,175.766,31.863,155.734
C06848=1074.333,385.728,395.369,175.761,31.856,155.733
C06849=1074.327,385.487,395.408,175.757,31.849,155.731
C06850=1074.320,385.245,395.446,175.753,31.842,155.730
C06851=1074.313,385.004,395.484,175.749,31.834,155.728
C06852=1074.307,384.762,395.523,175.745,31.827,155.727
C06853=1074.300,384.515,395.562,175.741,31.820,155.725
C06854=1074.293,384.269,395.602,175.737,31.812,155.724
C06855=1074.287,384.022,395.641,175.732,31.805,155.722
C06856=1074.280,383.775,395.680,175.728,31.798,155.721
C06857=1074.274,383.528,395.719,175.724,31.791,155.719
C06858=1074.267,383.281,395.758,175.720,31.784,155.718
C06859=1074.260,383.035,395.798,175.715,31.777,155.716
C06860=1074.254,382.788,395.837,175.711,31.769,155.715
C06861=1074.247,382.541,395.875,175.708,31.762,155.713
C06862=1074.240,382.294,395.914,175.703,31.755,155.712
C06863=1074.234,382.047,395.954,175.699,31.748,155.710
C06864=1074.228,381.801,395.992,175.695,31.740,155.709
C06865=1074.221,381.554,396.031,175.691,31.733,155.708
C06866=1074.214,381.307,396.070,175.687,31.727,155.706
C06867=1074.207,381.060,396.109,175.682,31.720,155.705
C06868=1074.200,380.814,396.147,175.679,31.713,155.703
C06869=1074.194,380.567,396.186,175.674,31.706,155.702
C06870=1074.187,380.319,396.224,175.670,31.699,155.700
C06871=1074.180,380.073,396.263,175.667,31.692,155.699
C06872=1074.173,379.826,396.302,175.662,31.685,155.698
C06873=1074.167,379.579,396.341,175.658,31.678,155.696
C06874=1074.160,379.332,396.380,175.654,31.671,155.695
C06875=1074.154,379.085,396.418,175.650,31.664,155.693
C06876=1074.147,378.839,396.456,175.646,31.657,155.692
C06877=1074.140,378.592,396.495,175.641,31.650,155.690
C06878=1074.133,378.345,396.534,175.638,31.643,155.689
C06879=1074.127,378.097,396.572,175.634,31.637,155.688
C06880=1074.121,377.851,396.611,175.629,31.630,155.686
C06881=1074.114,377.604,396.649,175.626,31.623,155.685
C06882=1074.107,377.357,396.687,175.622,31.616,155.683
C06883=1074.100,377.111,396.726,175.617,31.609,155.682
C06884=1074.093,376.863,396.764,175.614,31.602,155.681
C06885=1074.087,376.617,396.802,175.610,31.596,155.679
C06886=1074.081,376.369,396.841,175.605,31.589,155.678
C06887=1074.074,376.123,396.879,175.602,31.582,155.677
C06888=1074.068,375.876,396.917,175.598,31.576,155.675
C06889=1074.061,375.629,396.956,175.593,31.569,155.674
C06890=1074.055,375.382,396.994,175.590,31.562,155.672
C06891=1074.048,375.136,397.032,175.586,31.555,155.671
C06892=1074.041,374.888,397.070,175.582,31.549,155.670
C06893=1074.035,374.641,397.108,175.577,31.542,155.668
C06894=1074.028,374.395,397.147,175.574,31.535,155.667
C06895=1074.022,374.147,397.185,175.570,31.529,155.666
C06896=1074.015,373.900,397.223,175.565,31.522,155.664
C06897=1074.010,373.653,397.261,175.562,31.516,155.663
C06898=1074.002,373.407,397.299,175.558,31.509,155.662
C06899=1073.995,373.159,397.337,175.554,31.502,155.660
C06900=1073.990,372.912,397.375,175.550,31.496,155.659
C06901=1073.984,372.685,397.409,175.547,31.490,155.658
C06902=1073.977,372.459,397.445,175.543,31.484,155.657
C06903=1073.971,372.232,397.479,175.540,31.478,155.655
C06904=1073.965,372.004,397.514,175.536,31.472,155.654
C06905=1073.959,371.777,397.548,175.532,31.466,155.653
C06906=1073.953,371.550,397.584,175.529,31.460,155.652
C06907=1073.947,371.323,397.618,175.525,31.454,155.651
C06908=1073.941,371.096,397.653,175.521,31.448,155.649
C06909=1073.934,370.849,397.690,175.518,31.442,155.648
C06910=1073.928,370.602,397.728,175.514,31.435,155.647
C06911=1073.921,370.355,397.766,175.510,31.429,155.646
C06912=1073.915,370.108,397.803,175.506,31.423,155.644
C06913=1073.907,369.861,397.841,175.502,31.416,155.643
C06914=1073.902,369.614,397.879,175.498,31.410,155.642
C06915=1073.894,369.367,397.916,175.495,31.404,155.641
C06916=1073.888,369.120,397.954,175.490,31.397,155.639
C06917=1073.882,368.872,397.991,175.486,31.391,155.638
C06918=1073.876,368.626,398.029,175.483,31.385,155.637
C06919=1073.869,368.378,398.067,175.479,31.378,155.635
C06920=1073.862,368.132,398.104,175.475,31.372,155.634
C06921=1073.856,367.884,398.141,175.472,31.366,155.633
C06922=1073.850,367.638,398.178,175.467,31.359,155.632
C06923=1073.844,367.391,398.216,175.463,31.353,155.631
C06924=1073.836,367.144,398.254,175.460,31.347,155.629
C06925=1073.831,366.896,398.291,175.456,31.341,155.628
C06926=1073.824,366.649,398.328,175.452,31.335,155.627
C06927=1073.817,366.402,398.365,175.449,31.328,155.625
C06928=1073.811,366.155,398.402,175.444,31.322,155.624
C06929=1073.804,365.908,398.440,175.440,31.316,155.623
C06930=1073.798,365.661,398.477,175.437,31.310,155.622
C06931=1073.791,365.414,398.515,175.433,31.303,155.621
C06932=1073.786,365.166,398.552,175.429,31.297,155.619
C06933=1073.779,364.920,398.589,175.426,31.291,155.618
C06934=1073.772,364.672,398.626,175.422,31.285,155.617
C06935=1073.766,364.425,398.663,175.419,31.279,155.616
C06936=1073.760,364.178,398.700,175.414,31.273,155.615
C06937=1073.753,363.931,398.737,175.410,31.267,155.613
C06938=1073.747,363.684,398.774,175.407,31.261,155.612
C06939=1073.741,363.437,398.811,175.403,31.255,155.611
C06940=1073.734,363.189,398.848,175.399,31.249,155.610
C06941=1073.727,362.943,398.885,175.396,31.243,155.609
C06942=1073.721,362.696,398.921,175.392,31.237,155.607
C06943=1073.715,362.448,398.959,175.388,31.231,155.606
C06944=1073.708,362.200,398.995,175.385,31.225,155.605
C06945=1073.697,361.823,399.052,175.378,31.215,155.603
C06946=1073.688,361.445,399.108,175.373,31.206,155.602
C06947=1073.678,361.067,399.164,175.367,31.198,155.600
C06948=1073.669,360.689,399.220,175.362,31.189,155.598
C06949=1073.662,360.441,399.257,175.358,31.183,155.597
C06950=1073.655,360.194,399.294,175.355,31.177,155.596
C06951=1073.649,359.947,399.330,175.350,31.171,155.595
C06952=1073.643,359.700,399.367,175.346,31.165,155.593
C06953=1073.637,359.453,399.404,175.343,31.159,155.592
C06954=1073.630,359.205,399.440,175.339,31.153,155.591
C06955=1073.624,358.958,399.477,175.336,31.147,155.590
C06956=1073.617,358.711,399.513,175.332,31.141,155.589
C06957=1073.610,358.404,399.558,175.327,31.134,155.587
C06958=1073.601,358.098,399.603,175.323,31.127,155.586
C06959=1073.594,357.792,399.648,175.318,31.120,155.585
C06960=1073.586,357.484,399.693,175.314,31.113,155.583
C06961=1073.579,357.237,399.730,175.310,31.107,155.582
C06962=1073.573,356.990,399.766,175.307,31.101,155.581
C06963=1073.567,356.743,399.803,175.303,31.095,155.580
C06964=1073.561,356.496,399.838,175.299,31.090,155.579
C06965=1073.553,356.248,399.875,175.296,31.084,155.578
C06966=1073.547,356.001,399.911,175.292,31.078,155.576
C06967=1073.540,355.754,399.948,175.288,31.072,155.575
C06968=1073.534,355.506,399.983,175.285,31.066,155.574
C06969=1073.528,355.259,400.020,175.281,31.061,155.573
C06970=1073.522,355.012,400.056,175.278,31.056,155.572
C06971=1073.516,354.765,400.092,175.274,31.050,155.571
C06972=1073.509,354.518,400.128,175.270,31.044,155.570
C06973=1073.503,354.270,400.164,175.267,31.038,155.569
C06974=1073.497,354.023,400.201,175.263,31.033,155.568
C06975=1073.491,353.776,400.237,175.259,31.027,155.567
C06976=1073.484,353.528,400.272,175.256,31.021,155.566
C06977=1073.478,353.281,400.309,175.252,31.016,155.565
C06978=1073.472,353.034,400.344,175.249,31.010,155.563
C06979=1073.465,352.787,400.381,175.245,31.004,155.562
C06980=1073.459,352.539,400.416,175.242,30.999,155.561
C06981=1073.453,352.291,400.452,175.239,30.994,155.560
C06982=1073.446,352.045,400.488,175.235,30.988,155.559
C06983=1073.440,351.797,400.524,175.232,30.982,155.558
C06984=1073.434,351.550,400.560,175.228,30.977,155.557
C06985=1073.427,351.302,400.595,175.224,30.971,155.556
C06986=1073.421,351.055,400.631,175.221,30.966,155.555
C06987=1073.415,350.808,400.668,175.217,30.960,155.554
C06988=1073.408,350.560,400.703,175.213,30.955,155.553
C06989=1073.402,350.313,400.738,175.210,30.949,155.552
C06990=1073.396,350.065,400.774,175.206,30.944,155.551
C06991=1073.389,349.818,400.810,175.203,30.939,155.550
C06992=1073.383,349.571,400.846,175.199,30.933,155.549
C06993=1073.376,349.323,400.881,175.195,30.928,155.548
C06994=1073.370,349.076,400.916,175.193,30.922,155.547
C06995=1073.364,348.829,400.952,175.189,30.917,155.546
C06996=1073.358,348.581,400.987,175.186,30.911,155.545
C06997=1073.352,348.334,401.023,175.182,30.906,155.544
C06998=1073.345,348.086,401.059,175.178,30.900,155.543
C06999=1073.338,347.839,401.094,175.175,30.895,155.541
C07000=1073.332,347.591,401.130,175.171,30.889,155.540
C07001=1073.326,347.344,401.165,175.168,30.884,155.539
C07002=1073.320,347.097,401.201,175.164,30.878,155.538
C07003=1073.313,346.850,401.236,175.161,30.873,155.537
C07004=1073.307,346.602,401.271,175.158,30.868,155.536
C07005=1073.301,346.355,401.307,175.154,30.863,155.535
C07006=1073.295,346.107,401.342,175.151,30.857,155.534
C07007=1073.289,345.860,401.376,175.147,30.852,155.533
C07008=1073.283,345.612,401.412,175.143,30.846,155.532
C07009=1073.277,345.395,401.443,175.141,30.842,155.531
C07010=1073.272,345.179,401.475,175.137,30.837,155.531
C07011=1073.266,344.961,401.504,175.134,30.832,155.530
C07012=1073.261,344.745,401.536,175.132,30.828,155.529
C07013=1073.255,344.528,401.567,175.128,30.823,155.528
C07014=1073.250,344.311,401.597,175.125,30.819,155.527
C07015=1073.245,344.094,401.629,175.123,30.814,155.526
C07016=1073.239,343.877,401.659,175.119,30.809,155.525
C07017=1073.233,343.629,401.694,175.116,30.804,155.524
C07018=1073.226,343.382,401.730,175.113,30.799,155.523
C07019=1073.219,343.134,401.764,175.109,30.794,155.522
C07020=1073.214,342.887,401.799,175.106,30.788,155.521
C07021=1073.207,342.639,401.834,175.102,30.783,155.520
C07022=1073.201,342.391,401.869,175.099,30.778,155.519
C07023=1073.195,342.144,401.904,175.095,30.773,155.519
C07024=1073.189,341.897,401.939,175.092,30.768,155.517
C07025=1073.182,341.649,401.974,175.089,30.763,155.517
C07026=1073.175,341.402,402.009,175.085,30.758,155.516
C07027=1073.170,341.154,402.044,175.082,30.752,155.515
C07028=1073.163,340.907,402.079,175.078,30.747,155.514
C07029=1073.157,340.659,402.113,175.075,30.742,155.513
C07030=1073.151,340.412,402.148,175.072,30.737,155.512
C07031=1073.145,340.164,402.183,175.068,30.731,155.511
C07032=1073.139,339.917,402.218,175.065,30.726,155.510
C07033=1073.132,339.669,402.252,175.062,30.722,155.509
C07034=1073.126,339.422,402.287,175.058,30.716,155.508
C07035=1073.121,339.174,402.322,175.055,30.711,155.507
C07036=1073.114,338.926,402.356,175.051,30.706,155.506
C07037=1073.108,338.679,402.391,175.048,30.701,155.505
C07038=1073.101,338.431,402.425,175.045,30.696,155.504
C07039=1073.095,338.184,402.461,175.041,30.691,155.503
C07040=1073.090,337.937,402.495,175.038,30.685,155.502
C07041=1073.083,337.689,402.530,175.034,30.680,155.501
C07042=1073.077,337.441,402.564,175.032,30.675,155.500
C07043=1073.070,337.194,402.599,175.028,30.670,155.499
C07044=1073.064,336.946,402.633,175.024,30.665,155.499
C07045=1073.058,336.699,402.667,175.021,30.660,155.498
C07046=1073.052,336.451,402.702,175.018,30.655,155.497
C07047=1073.046,336.203,402.736,175.015,30.650,155.496
C07048=1073.039,335.956,402.771,175.011,30.645,155.495
C07049=1073.033,335.709,402.805,175.008,30.640,155.494
C07050=1073.027,335.461,402.839,175.005,30.635,155.493
C07051=1073.021,335.213,402.873,175.001,30.630,155.492
C07052=1073.014,334.965,402.908,174.998,30.625,155.491
C07053=1073.009,334.718,402.942,174.995,30.621,155.490
C07054=1073.002,334.470,402.976,174.991,30.616,155.489
C07055=1072.996,334.223,403.010,174.988,30.611,155.488
C07056=1072.990,333.975,403.045,174.985,30.606,155.487
C07057=1072.984,333.728,403.079,174.982,30.601,155.487
C07058=1072.977,333.480,403.113,174.978,30.596,155.486
C07059=1072.972,333.232,403.147,174.975,30.591,155.485
C07060=1072.965,332.984,403.182,174.972,30.586,155.484
C07061=1072.959,332.737,403.216,174.968,30.581,155.483
C07062=1072.953,332.490,403.250,174.965,30.576,155.482
C07063=1072.946,332.242,403.284,174.962,30.571,155.481
C07064=1072.940,331.995,403.318,174.959,30.566,155.480
C07065=1072.935,331.774,403.348,174.956,30.562,155.479
C07066=1072.930,331.556,403.378,174.952,30.557,155.479
C07067=1072.924,331.336,403.408,174.950,30.553,155.478
C07068=1072.919,331.117,403.438,174.947,30.549,155.477
C07069=1072.913,330.897,403.468,174.944,30.544,155.476
C07070=1072.907,330.677,403.499,174.941,30.540,155.475
C07071=1072.902,330.458,403.528,174.938,30.536,155.475
C07072=1072.896,330.238,403.558,174.936,30.532,155.474
C07073=1072.890,329.991,403.592,174.932,30.527,155.473
C07074=1072.883,329.743,403.626,174.929,30.522,155.472
C07075=1072.877,329.496,403.660,174.926,30.517,155.471
C07076=1072.871,329.247,403.694,174.922,30.512,155.471
C07077=1072.865,329.000,403.727,174.920,30.508,155.470
C07078=1072.859,328.753,403.761,174.916,30.503,155.469
C07079=1072.852,328.505,403.794,174.912,30.498,155.468
C07080=1072.846,328.257,403.828,174.910,30.494,155.467
C07081=1072.840,328.009,403.862,174.906,30.489,155.466
C07082=1072.833,327.762,403.895,174.903,30.484,155.465
C07083=1072.828,327.514,403.929,174.900,30.479,155.465
C07084=1072.820,327.266,403.963,174.897,30.474,155.464
C07085=1072.815,327.018,403.996,174.894,30.470,155.463
C07086=1072.808,326.771,404.029,174.890,30.465,155.462
C07087=1072.802,326.523,404.063,174.887,30.461,155.461
C07088=1072.796,326.275,404.097,174.884,30.456,155.460
C07089=1072.790,326.028,404.130,174.881,30.451,155.459
C07090=1072.784,325.780,404.164,174.877,30.446,155.459
C07091=1072.777,325.532,404.197,174.874,30.441,155.458
C07092=1072.771,325.285,404.231,174.871,30.437,155.457
C07093=1072.765,325.037,404.264,174.868,30.432,155.456
C07094=1072.759,324.789,404.297,174.865,30.428,155.455
C07095=1072.752,324.542,404.331,174.861,30.422,155.454
C07096=1072.747,324.294,404.364,174.859,30.418,155.453
C07097=1072.740,324.046,404.397,174.855,30.413,155.453
C07098=1072.735,323.799,404.431,174.852,30.409,155.452
C07099=1072.728,323.551,404.464,174.849,30.404,155.451
C07100=1072.722,323.303,404.498,174.846,30.399,155.450
C07101=1072.716,323.055,404.530,174.843,30.394,155.449
C07102=1072.710,322.808,404.564,174.839,30.390,155.448
C07103=1072.704,322.560,404.597,174.836,30.386,155.448
C07104=1072.698,322.312,404.630,174.833,30.381,155.447
C07105=1072.692,322.065,404.663,174.830,30.376,155.446
C07106=1072.685,321.816,404.696,174.827,30.371,155.445
C07107=1072.679,321.569,404.730,174.824,30.367,155.444
C07108=1072.673,321.322,404.763,174.821,30.362,155.443
C07109=1072.667,321.074,404.796,174.817,30.357,155.443
C07110=1072.661,320.826,404.829,174.814,30.353,155.442
C07111=1072.655,320.578,404.863,174.811,30.348,155.441
C07112=1072.649,320.331,404.895,174.808,30.344,155.440
C07113=1072.644,320.083,404.929,174.805,30.339,155.439
C07114=1072.637,319.835,404.961,174.802,30.334,155.438
C07115=1072.631,319.588,404.994,174.799,30.330,155.438
C07116=1072.625,319.340,405.027,174.796,30.325,155.437
C07117=1072.619,319.092,405.060,174.792,30.320,155.436
C07118=1072.614,318.844,405.094,174.790,30.315,155.435
C07119=1072.607,318.597,405.126,174.786,30.311,155.434
C07120=1072.601,318.349,405.159,174.784,30.307,155.433
C07121=1072.595,318.126,405.189,174.780,30.302,155.433
C07122=1072.590,317.903,405.218,174.778,30.298,155.432
C07123=1072.585,317.680,405.248,174.775,30.294,155.431
C07124=1072.579,317.458,405.278,174.772,30.290,155.430
C07125=1072.574,317.236,405.308,174.770,30.286,155.430
C07126=1072.568,317.013,405.337,174.767,30.281,155.429
C07127=1072.564,316.790,405.367,174.764,30.278,155.428
C07128=1072.558,316.567,405.396,174.761,30.273,155.428
C07129=1072.552,316.319,405.428,174.758,30.269,155.427
C07130=1072.546,316.071,405.461,174.755,30.264,155.426
C07131=1072.541,315.824,405.494,174.752,30.259,155.425
C07132=1072.534,315.577,405.527,174.750,30.255,155.424
C07133=1072.528,315.329,405.560,174.746,30.251,155.424
C07134=1072.523,315.080,405.592,174.744,30.246,155.423
C07135=1072.517,314.833,405.625,174.740,30.241,155.422
C07136=1072.510,314.585,405.658,174.737,30.237,155.421
C07137=1072.505,314.337,405.690,174.734,30.232,155.420
C07138=1072.498,314.089,405.722,174.731,30.228,155.419
C07139=1072.492,313.842,405.755,174.728,30.223,155.419
C07140=1072.486,313.594,405.787,174.725,30.219,155.418
C07141=1072.479,313.346,405.820,174.722,30.214,155.417
C07142=1072.473,313.098,405.852,174.719,30.210,155.416
C07143=1072.467,312.850,405.885,174.715,30.206,155.416
C07144=1072.461,312.603,405.918,174.713,30.201,155.415
C07145=1072.455,312.354,405.950,174.709,30.197,155.414
C07146=1072.449,312.107,405.982,174.707,30.192,155.413
C07147=1072.442,311.859,406.014,174.703,30.188,155.412
C07148=1072.436,311.612,406.046,174.701,30.183,155.412
C07149=1072.430,311.364,406.078,174.697,30.179,155.411
C07150=1072.424,311.116,406.110,174.694,30.175,155.410
C07151=1072.418,310.868,406.143,174.691,30.171,155.409
C07152=1072.412,310.620,406.175,174.688,30.166,155.409
C07153=1072.406,310.372,406.208,174.686,30.162,155.408
C07154=1072.399,310.124,406.239,174.682,30.157,155.407
C07155=1072.393,309.876,406.271,174.680,30.153,155.406
C07156=1072.387,309.629,406.303,174.676,30.148,155.406
C07157=1072.381,309.381,406.336,174.673,30.144,155.405
C07158=1072.375,309.133,406.368,174.670,30.140,155.404
C07159=1072.368,308.885,406.400,174.667,30.136,155.403
C07160=1072.362,308.637,406.432,174.664,30.131,155.403
C07161=1072.357,308.390,406.463,174.661,30.127,155.402
C07162=1072.351,308.142,406.496,174.659,30.122,155.401
C07163=1072.345,307.894,406.528,174.655,30.118,155.400
C07164=1072.338,307.646,406.560,174.652,30.113,155.399
C07165=1072.332,307.398,406.592,174.649,30.109,155.399
C07166=1072.326,307.151,406.624,174.646,30.105,155.398
C07167=1072.320,306.903,406.656,174.643,30.100,155.397
C07168=1072.313,306.655,406.687,174.640,30.096,155.396
C07169=1072.308,306.407,406.719,174.638,30.092,155.396
C07170=1072.302,306.159,406.751,174.634,30.087,155.395
C07171=1072.296,305.911,406.783,174.632,30.083,155.394
C07172=1072.290,305.664,406.815,174.628,30.079,155.393
C07173=1072.284,305.416,406.847,174.625,30.074,155.393
C07174=1072.278,305.168,406.879,174.623,30.070,155.392
C07175=1072.272,304.920,406.911,174.619,30.065,155.391
C07176=1072.266,304.672,406.942,174.617,30.061,155.390
C07177=1072.260,304.451,406.970,174.614,30.057,155.390
C07178=1072.255,304.230,406.999,174.612,30.053,155.389
C07179=1072.249,304.009,407.027,174.609,30.050,155.388
C07180=1072.244,303.788,407.056,174.606,30.046,155.388
C07181=1072.239,303.567,407.084,174.604,30.042,155.387
C07182=1072.234,303.346,407.112,174.601,30.038,155.386
C07183=1072.229,303.125,407.140,174.599,30.034,155.386
C07184=1072.223,302.904,407.169,174.596,30.030,155.385
C07185=1072.217,302.657,407.200,174.592,30.026,155.384
C07186=1072.211,302.408,407.231,174.590,30.022,155.383
C07187=1072.205,302.160,407.264,174.587,30.018,155.383
C07188=1072.199,301.913,407.295,174.584,30.013,155.382
C07189=1072.193,301.665,407.327,174.581,30.009,155.381
C07190=1072.188,301.417,407.358,174.579,30.004,155.381
C07191=1072.181,301.169,407.390,174.575,30.000,155.380
C07192=1072.176,300.922,407.421,174.572,29.996,155.379
C07193=1072.170,300.673,407.453,174.570,29.992,155.378
C07194=1072.164,300.426,407.484,174.566,29.987,155.378
C07195=1072.158,300.178,407.516,174.564,29.983,155.377
C07196=1072.153,299.930,407.547,174.561,29.979,155.376
C07197=1072.146,299.682,407.579,174.558,29.974,155.375
C07198=1072.141,299.434,407.610,174.555,29.970,155.375
C07199=1072.135,299.186,407.642,174.553,29.965,155.374
C07200=1072.129,298.939,407.673,174.549,29.961,155.373
C07201=1072.123,298.690,407.704,174.547,29.957,155.372
C07202=1072.118,298.442,407.736,174.544,29.953,155.372
C07203=1072.111,298.194,407.767,174.541,29.948,155.371
C07204=1072.106,297.946,407.798,174.538,29.944,155.370
C07205=1072.099,297.698,407.830,174.535,29.940,155.369
C07206=1072.094,297.451,407.861,174.532,29.935,155.369
C07207=1072.087,297.202,407.892,174.529,29.931,155.368
C07208=1072.082,296.955,407.924,174.527,29.927,155.367
C07209=1072.076,296.706,407.954,174.523,29.922,155.366
C07210=1072.069,296.459,407.985,174.521,29.919,155.366
C07211=1072.064,296.210,408.017,174.518,29.914,155.365
C07212=1072.058,295.963,408.048,174.515,29.910,155.364
C07213=1072.052,295.715,408.078,174.512,29.906,155.364
C07214=1072.046,295.467,408.110,174.509,29.902,155.363
C07215=1072.040,295.219,408.141,174.507,29.897,155.362
C07216=1072.033,294.971,408.172,174.503,29.893,155.361
C07217=1072.028,294.723,408.203,174.501,29.889,155.361
C07218=1072.022,294.475,408.234,174.498,29.885,155.360
C07219=1072.016,294.227,408.265,174.495,29.881,155.359
C07220=1072.009,293.979,408.295,174.492,29.877,155.359
C07221=1072.004,293.731,408.327,174.490,29.872,155.358
C07222=1071.997,293.483,408.358,174.487,29.868,155.357
C07223=1071.992,293.235,408.388,174.484,29.864,155.356
C07224=1071.986,292.988,408.419,174.481,29.860,155.356
C07225=1071.980,292.739,408.451,174.478,29.856,155.355
C07226=1071.974,292.491,408.481,174.475,29.851,155.354
C07227=1071.968,292.243,408.511,174.472,29.847,155.353
C07228=1071.961,291.995,408.543,174.470,29.843,155.353
C07229=1071.956,291.748,408.573,174.467,29.839,155.352
C07230=1071.950,291.499,408.604,174.464,29.835,155.351
C07231=1071.944,291.251,408.635,174.461,29.830,155.351
C07232=1071.938,291.004,408.666,174.459,29.826,155.350
C07233=1071.933,290.790,408.692,174.456,29.823,155.349
C07234=1071.928,290.576,408.718,174.453,29.819,155.349
C07235=1071.922,290.362,408.745,174.451,29.815,155.348
C07236=1071.917,290.148,408.771,174.449,29.812,155.348
C07237=1071.913,289.936,408.798,174.447,29.808,155.347
C07238=1071.907,289.722,408.824,174.444,29.805,155.346
C07239=1071.901,289.508,408.850,174.441,29.801,155.346
C07240=1071.897,289.294,408.877,174.439,29.797,155.345
C07241=1071.891,289.046,408.907,174.436,29.794,155.344
C07242=1071.885,288.799,408.938,174.434,29.790,155.344
C07243=1071.879,288.550,408.968,174.431,29.785,155.343
C07244=1071.873,288.302,408.999,174.429,29.781,155.342
C07245=1071.867,288.054,409.029,174.425,29.777,155.342
C07246=1071.861,287.806,409.060,174.423,29.773,155.341
C07247=1071.855,287.558,409.090,174.420,29.769,155.340
C07248=1071.849,287.310,409.121,174.417,29.765,155.340
C07249=1071.843,287.062,409.151,174.414,29.761,155.339
C07250=1071.837,286.814,409.182,174.411,29.757,155.338
C07251=1071.831,286.566,409.212,174.409,29.753,155.337
C07252=1071.824,286.318,409.242,174.406,29.748,155.337
C07253=1071.818,286.069,409.272,174.404,29.744,155.336
C07254=1071.813,285.822,409.302,174.400,29.740,155.335
C07255=1071.807,285.574,409.332,174.398,29.736,155.335
C07256=1071.800,285.325,409.363,174.395,29.732,155.334
C07257=1071.795,285.077,409.394,174.393,29.728,155.333
C07258=1071.789,284.830,409.424,174.390,29.724,155.333
C07259=1071.783,284.581,409.453,174.386,29.720,155.332
C07260=1071.777,284.333,409.484,174.384,29.716,155.331
C07261=1071.771,284.085,409.515,174.381,29.711,155.330
C07262=1071.765,283.837,409.545,174.379,29.708,155.330
C07263=1071.759,283.589,409.575,174.376,29.704,155.329
C07264=1071.753,283.341,409.604,174.373,29.699,155.328
C07265=1071.747,283.093,409.635,174.370,29.695,155.328
C07266=1071.741,282.845,409.665,174.368,29.691,155.327
C07267=1071.735,282.596,409.695,174.365,29.687,155.326
C07268=1071.729,282.348,409.725,174.363,29.683,155.326
C07269=1071.724,282.101,409.756,174.359,29.679,155.325
C07270=1071.718,281.852,409.785,174.357,29.674,155.324
C07271=1071.712,281.605,409.815,174.354,29.671,155.324
C07272=1071.706,281.357,409.845,174.352,29.667,155.323
C07273=1071.700,281.108,409.875,174.349,29.662,155.322
C07274=1071.694,280.860,409.906,174.346,29.658,155.322
C07275=1071.688,280.611,409.935,174.343,29.654,155.321
C07276=1071.683,280.364,409.966,174.340,29.650,155.320
C07277=1071.676,280.115,409.995,174.338,29.646,155.319
C07278=1071.670,279.868,410.025,174.335,29.642,155.319
C07279=1071.665,279.619,410.055,174.333,29.638,155.318
C07280=1071.658,279.372,410.085,174.330,29.634,155.317
C07281=1071.652,279.122,410.115,174.328,29.630,155.317
C07282=1071.646,278.875,410.145,174.324,29.626,155.316
C07283=1071.640,278.627,410.174,174.322,29.622,155.315
C07284=1071.634,278.379,410.204,174.319,29.618,155.315
